# B&R Automation Studio project Agroittica (part 5)

#### Cyclic.st
```iecst
PROGRAM _CYCLIC

	//data to write
	kgb:=0;

	FOR kgb := 0 TO kgb < 30 DO
		rpt_row[kgb]:= 1;
	END_FOR;

	IF (NOT glb_data.Trigger) THEN  rpt_write_req := 0; END_IF

	IF (fucking_debug) THEN step_rpt := step_force; END_IF

	//comando reset progressivo
	IF (struct_time.day <> Saved_day (*Day_test<> Saved_day*)) THEN
		Counter_Reset := 1;
	END_IF;

	CASE step_rpt OF (* Stato di idle *)
		WAIT:
			TP_01.IN := 0;
			IF (glb_data.Trigger AND (NOT rpt_write_req))THEN

				xxx 				:= 0;
				step_rpt 			:= CHECK_FILES_NAME;
				rpt_write_req 		:= 1;				// Resetto la richiesta di scrittura del report
				glb_data.Trigger 	:= 0;			// Machine Cycle done Trigger reset;

				TP_01.IN := 1;

			END_IF
		ERROR:

			IF (glb_data.Trigger AND (NOT rpt_write_req))THEN

				xxx 				:= 0;
				step_rpt 			:= CHECK_FILES_NAME;
				rpt_write_req 		:= 1;				// Resetto la richiesta di scrittura del report
				glb_data.Trigger 	:= 0;			// Machine Cycle done Trigger reset;

			END_IF

		CHECK_FILES_NAME:	// GUARDO SE IL FILE CREATO E' LO STESSO DEL MASTER

			step_rpt := CREATE_FILE_NAME;

		CREATE_FILE_NAME: 	// CREO IL NOME DEI FILE

			memset (ADR(FileCreate_01),         0, SIZEOF(FileCreate_01)	);
			memset (ADR(FileWrite_01),          0, SIZEOF(FileWrite_01) 	);
			memset (ADR(FileClose_01),          0, SIZEOF(FileClose_01) 	);
			memset (ADR(FileCreate_03),         0, SIZEOF(FileCreate_03)    );
			memset (ADR(FileOpen_03),           0, SIZEOF(FileOpen_03)      );
			memset (ADR(FileWrite_03),          0, SIZEOF(FileWrite_03)     );
			memset (ADR(FileClose_03),          0, SIZEOF(FileClose_03)		);
			memset (ADR(string_rpt),			0, SIZEOF(string_rpt)		);
			memset (ADR(nome_file_doc),			0, SIZEOF(nome_file_doc)	);
			memset (ADR(nome_file_csv),			0, SIZEOF(nome_file_csv)	);
			memset (ADR(support_str),			0, SIZEOF(support_str)		);
			offset 		:= 0;

			(* Trasferisco nella struttura support_str l'orario attuale *)
			DT_TO_DTStructure(glb_time, ADR(struct_time));

			(* Genero il nome del file con la data odierna formato YYYY-MM-DD *)

			// inserimento anno nel nome del file
			memset (ADR(support_str), 0, SIZEOF(support_str));
			itoa(struct_time.year, ADR(support_str));
			strcpy(ADR(nome_file_doc), ADR(support_str));
			strcat(ADR(nome_file_doc), ADR(space));

			// inserimento mese nel nome del file
			memset (ADR(support_str), 0, SIZEOF(support_str));
			itoa(struct_time.month, ADR(support_str));
			IF (strlen(ADR(support_str)) = 1) THEN strcat(ADR(nome_file_doc), ADR("0")); END_IF;
			strcat(ADR(nome_file_doc), ADR(support_str));
			strcat(ADR(nome_file_doc), ADR(space));

			// inserimento giorno nel nome del file
			memset (ADR(support_str), 0, SIZEOF(support_str));
			itoa(struct_time.day, ADR(support_str));
			(*itoa(Day_test, ADR(support_str));*)
			IF (strlen(ADR(support_str)) = 1) THEN strcat(ADR(nome_file_doc), ADR("0")); END_IF;
			strcat(ADR(nome_file_doc), ADR(support_str));
			strcat(ADR(nome_file_doc), ADR(space));

			//Reset del numero progressivo quando cambia giorno
			IF Counter_Reset THEN
				Counter := 0;
				Counter_Reset := 0;
			END_IF;

			//inserimento del numero progressivo alla fine del nome del file csv
			memset (ADR(support_str), 0, SIZEOF(support_str));
			itoa(Counter, ADR(support_str));
			IF (strlen(ADR(support_str)) = 1) THEN strcat(ADR(nome_file_doc), ADR("0")); END_IF;
			strcat(ADR(nome_file_doc), ADR(support_str));

			strcpy(ADR(nome_file_csv), ADR(nome_file_doc));
			strcat(ADR(nome_file_csv), ADR(estensione));				// creo il file YYYY-MM-DD.csv

			step_rpt := CREATE_CSV_FILE;

		CREATE_CSV_FILE: // CREO IL FILE .CSV

			FileCreate_03.enable  := 1;
			FileCreate_03.pDevice := ADR(DATA);
			FileCreate_03.pFile   := ADR(nome_file_csv);

			FileCreate_03;

			IF (FileCreate_03.status = 0) THEN

				offset 					:= 0;
				step_rpt   				:= OPEN_CSV_FILE;
				FileCreate_03.enable 	:= 0;
				RowCounterFile			:= 0;

			ELSIF (FileCreate_03.status = 20705) THEN (* file già esistente *)
				step_rpt 				:= OPEN_CSV_FILE;
				FileCreate_03.enable 	:= 0;
			END_IF

		OPEN_CSV_FILE: // APRO IL FILE CSV

			FileOpen_03.enable    := 1;
			FileOpen_03.pDevice   := ADR(DATA);
			FileOpen_03.pFile     := ADR(nome_file_csv);
			FileOpen_03.mode      := FILE_RW;

			FileOpen_03;

			IF (FileOpen_03.status = 0) THEN

				step_rpt := CREATE_HEADER_CSV_FILE;

				memset (ADR(string_rpt), 	0, SIZEOF(string_rpt)	);
				memset (ADR(support_str),   0, SIZEOF(support_str)  );

				ident_csv			:= FileOpen_03.ident;
				FileOpen_03.enable 	:= 0;
				filelen := FileOpen_03.filelen;

			ELSIF (FileOpen_03.status <> 65535) THEN

				step_rpt	 		:= ERROR;
				numero_errore   	:= FileIoGetSysError();
				FileOpen_03.enable 	:= 0;
			END_IF

			// salvo il giorno in una variabile ritentiva
			Saved_day := struct_time.day;
			//Saved_day := Day_test;

			//Gestione numero progressivo, ogni 400000 elementi il progressivo avanza
			IF (filelen >= 400000) THEN
				New_CSV := 1;
			ELSE
				New_CSV := 0;
			END_IF;

			IF (New_CSV AND (NOT New_CSV_cmd)) THEN
				Counter 	:= Counter +1;
				New_CSV_cmd := 1;
			ELSIF ((NOT New_CSV) AND New_CSV_cmd) THEN
				New_CSV_cmd := 0;
			END_IF;

		CREATE_HEADER_CSV_FILE:

			// Il file è vuoto
			IF (filelen < 101) THEN //lunghezza della intestazione

				memset (ADR(string_rpt), 0, SIZEOF(string_rpt));
				// HEADER CDV FILE -------------------------------------------------------------------
				// Salvo l'intestazione di 120 caratteri

				//	sep:=;
				//	Report
				//	Dati misurazione particolari
				//	Mould Code := jhgfdsasdfghj;
				//
				//	Timestamp;Recipe Name;QRCode;Dato 1;Dato 2;Dato 3;Dato 4;Dato 5;Dato 6;Dato 7;Dato 8;Code;Material type;Material Color;Mould Code;Density;Volume;Peso;Temperature;Peso inserto;\n
				//  Timestamp;Recipe Name;QRCode;Dato 1;Dato 2;Dato 3;Dato 4;Dato 5;Dato 6;Dato 7;Dato 8;Code;Material type;Material Color;Mould Code;Density;Volume;Peso;Temperature;Peso inserto;\n
				//  012345678901234567890123456789012345678901234567890123456789012345678901234567890123456789012345678901234567890123456789
				//	0_________1_________2_________3_________4_________5_________6_________7_________8_________9_________10________11________

				strcpy(ADR(string_rpt), ADR('sep:=;$r$nReport$r$nDati misurazione particolari$r$n$r$n'));
				strcat(ADR(string_rpt), ADR('$r$n'));
				strcat(ADR(string_rpt), ADR('TIMESTAMP;BILANCIA;SENSORE PISTOLA;PISTONE SOLLEVAMENTO SU;PISTONE SOLLEVAMENTO GIU;PISTOLA 1;PISTOLA 2;'));
				strcat(ADR(string_rpt), ADR('$r$n'));
				// END HEADER ------------------------------------------------------------------------

				// TIMESTAMP
				memset (ADR(support_str), 0, SIZEOF(support_str));
				ascDT(glb_data.time_stamp[xxx],ADR(support_str),SIZEOF(support_str));
				IF (strlen(ADR(support_str)) = 1) THEN strcat(ADR(string_rpt), ADR('0')); END_IF
				strcat(ADR(string_rpt), ADR(support_str));
				strcat(ADR(string_rpt), ADR(';'));

				// BILANCIA
				memset (ADR(support_str), 0, SIZEOF(support_str));
				strcat(ADR(string_rpt), ADR(glb_data.bilancia[xxx]));
				strcat(ADR(string_rpt), ADR(';'));

				// SENSORE PISTOLA
				memset (ADR(support_str), 0, SIZEOF(support_str));
				itoa(glb_data.sensore_pistola[xxx], ADR(support_str));
				strcat(ADR(string_rpt), ADR(support_str));
				strcat(ADR(string_rpt), ADR(';'));

				// PISTONE SOLLEVAMENTO SU
				memset (ADR(support_str), 0, SIZEOF(support_str));
				itoa(glb_data.pistone_soll_su[xxx], ADR(support_str));
				strcat(ADR(string_rpt), ADR(support_str));
				strcat(ADR(string_rpt), ADR(';'));

				// PISTONE SOLLEVAMENTO GIU
				memset (ADR(support_str), 0, SIZEOF(support_str));
				itoa(glb_data.pistone_soll_giu[xxx], ADR(support_str));
				strcat(ADR(string_rpt), ADR(support_str));
				strcat(ADR(string_rpt), ADR(';'));

				// PISTOLA 1
				memset (ADR(support_str), 0, SIZEOF(support_str));
				itoa(glb_data.pistone_pistola_1[xxx], ADR(support_str));
				strcat(ADR(string_rpt), ADR(support_str));
				strcat(ADR(string_rpt), ADR(';'));

				// PISTOLA 2
				memset (ADR(support_str), 0, SIZEOF(support_str));
				itoa(glb_data.pistone_pistola_2[xxx], ADR(support_str));
				strcat(ADR(string_rpt), ADR(support_str));
				strcat(ADR(string_rpt), ADR(';'));

				strcat(ADR(string_rpt), ADR('$r$n'));

				filelen := 0;
				str_lenght := strlen(ADR(string_rpt)); (* restituisce la lunghezza della stringa senza terminatore nullo *)

				(* Preparo la struttura per la funzione di scrittura *)
				FileWrite_03.enable   := 1;
				FileWrite_03.ident    := ident_csv;
				FileWrite_03.offset   := filelen;
				FileWrite_03.pSrc     := ADR(string_rpt);
				FileWrite_03.len      := str_lenght;
				offset                := SIZEOF(USINT) * 240;

				RowCounterFile		  := 2; //2 ROWS * 110 BYTES
				filelen := filelen + str_lenght;

				step_rpt := WRITE_CSV_FILE;

			ELSIF (filelen > 102) THEN // Il file è già stato scritto

				memset (ADR(string_rpt), 0, SIZEOF(string_rpt));

				// TIMESTAMP
				memset (ADR(support_str), 0, SIZEOF(support_str));
				ascDT(glb_data.time_stamp[xxx],ADR(support_str),SIZEOF(support_str));
				IF (strlen(ADR(support_str)) = 1) THEN strcat(ADR(string_rpt), ADR('0')); END_IF
				strcat(ADR(string_rpt), ADR(support_str));
				strcat(ADR(string_rpt), ADR(';'));

				// BILANCIA
				memset (ADR(support_str), 0, SIZEOF(support_str));
				strcat(ADR(string_rpt), ADR(glb_data.bilancia[xxx]));
				strcat(ADR(string_rpt), ADR(';'));

				// SENSORE PISTOLA
				memset (ADR(support_str), 0, SIZEOF(support_str));
				itoa(glb_data.sensore_pistola[xxx], ADR(support_str));
				strcat(ADR(string_rpt), ADR(support_str));
				strcat(ADR(string_rpt), ADR(';'));

				// PISTONE SOLLEVAMENTO SU 1
				memset (ADR(support_str), 0, SIZEOF(support_str));
				itoa(glb_data.pistone_soll_su[xxx], ADR(support_str));
				strcat(ADR(string_rpt), ADR(support_str));
				strcat(ADR(string_rpt), ADR(';'));

				// PISTONE SOLLEVAMENTO GIU 1
				memset (ADR(support_str), 0, SIZEOF(support_str));
				itoa(glb_data.pistone_soll_giu[xxx], ADR(support_str));
				strcat(ADR(string_rpt), ADR(support_str));
				strcat(ADR(string_rpt), ADR(';'));

				// PISTOLA 1
				memset (ADR(support_str), 0, SIZEOF(support_str));
				itoa(glb_data.pistone_pistola_1[xxx], ADR(support_str));
				strcat(ADR(string_rpt), ADR(support_str));
				strcat(ADR(string_rpt), ADR(';'));

				// PISTOLA 2
				memset (ADR(support_str), 0, SIZEOF(support_str));
				itoa(glb_data.pistone_pistola_2[xxx], ADR(support_str));
				strcat(ADR(string_rpt), ADR(support_str));
				strcat(ADR(string_rpt), ADR(';'));

				strcat(ADR(string_rpt), ADR('$r$n'));

				RowCounterFile := RowCounterFile + 1;
//				filelen := RowCounterFile * 120;
//				filelen := FileOpen_03.filelen;

				str_lenght := strlen(ADR(string_rpt)); (* restituisce la lunghezza della stringa senza terminatore nullo *)

				(* Preparo la struttura per la funzione di scrittura *)
				FileWrite_03.enable   := 1;
				FileWrite_03.ident    := ident_csv;
				FileWrite_03.offset   := filelen;
				FileWrite_03.pSrc     := ADR(string_rpt);
				FileWrite_03.len      := str_lenght;
				offset                := offset + (SIZEOF(USINT) * 120);

				filelen := filelen + str_lenght;

				step_rpt := WRITE_CSV_FILE;

			ELSE  // Chiamato dal controllo densità con numero di ciclo a 0

				step_rpt := CLOSE_CSV_FILE;
			END_IF

		WRITE_CSV_FILE:

			FileWrite_03;

			IF (FileWrite_03.status = 0) THEN
				glb_data.Report_recorded 		:= 1;
				step_rpt 						:= CLOSE_CSV_FILE;
				FileWrite_03.enable 		  	:= 0;

				IF (xxx < 199) THEN
					xxx := xxx + 1;
					step_rpt 			:= CREATE_HEADER_CSV_FILE;

					//					glb_data.Trigger := 0;
				END_IF

			ELSIF (FileWrite_03.status <> 65535) THEN

				step_rpt	 		:= CLOSE_CSV_FILE;
				numero_errore   	:= FileIoGetSysError();
				FileWrite_03.enable := 0;
			END_IF

		CLOSE_CSV_FILE:

			FileClose_03.enable := 1;
			FileClose_03.ident  := ident_csv;
			FileClose_03;

			IF (FileClose_03.status = 0) THEN

//				step_rpt 				:= WAIT;
				FileClose_03.enable := 0;

			ELSIF (FileClose_03.status = 20721) THEN
				step_rpt 				:= WAIT;
				FileClose_03.enable := 0;

//				glb_data.Trigger := 1;

//				IF (xxx < 199) THEN
//					xxx := xxx + 1;
//					step_rpt 			:= OPEN_CSV_FILE;
//
////					glb_data.Trigger := 0;
//				END_IF

			ELSIF (FileClose_03.status <> 65535 AND FileClose_03.status <> 65534) THEN

				step_rpt	 		:= ERROR;

				numero_errore   	:= FileIoGetSysError();
				FileClose_03.enable := 0;
			END_IF

	END_CASE;

	(*********************************************** CREATE DIR WHERE SAVE THE CAVITIES INFO LINKE TO THE RECIPES **************************************************)

	IF ((DirCreate_05.status = 0) OR (DirCreate_05.status = 20725)) THEN	    (* IF status ok (0) OR dir already exists (20725)		 	*)
		DirCreate_05.enable 	:= 0;
	END_IF

	TP_01;

END_PROGRAM
```

#### Init.st
```iecst
PROGRAM _INIT
	(*/* Pulisco la memoria */*)

	memset (ADR(DirCreate_03),			 0, SIZEOF(DirCreate_03)   	 );
	memset (ADR(DirCreate_05),			 0, SIZEOF(DirCreate_05)   	 );
	memset (ADR(FileCreate_01),          0, SIZEOF(FileCreate_01)  	 );
	memset (ADR(FileCreate_03),          0, SIZEOF(FileCreate_03)  	 );
	memset (ADR(FileOpen_03),            0, SIZEOF(FileOpen_03)    	 );
	memset (ADR(FileWrite_01),           0, SIZEOF(FileWrite_01)   	 );
	memset (ADR(FileWrite_03),           0, SIZEOF(FileWrite_03)   	 );
	memset (ADR(FileClose_01),           0, SIZEOF(FileClose_01)	 );
	memset (ADR(FileClose_03),           0, SIZEOF(FileClose_03)	 );
	memset (ADR(string_rpt),			 0, SIZEOF(string_rpt)	 	 );
	memset (ADR(support_str),			 0, SIZEOF(support_str)  	 );

	step_rpt 			 := WAIT;
	RowCounterFile		 := 0;

	DirCreate_03.enable  := 1;
	DirCreate_03.pDevice := ADR(CF);
	DirCreate_03.pName   := ADR(DATA);

	DirCreate_03;

	IF ((DirCreate_03.status = 0) OR  (DirCreate_03.status = 20725)) THEN	    (*/* IF status ok (0) OR dir already exists (20725)			*/*)

		//DirCreate_03.status := 0;												(*/* set status ok											*/*)
	END_IF

	DirCreate_05.enable  := 1;
	DirCreate_05.pDevice := ADR(CF);
	DirCreate_05.pName   := ADR(CFG);

	DirCreate_05;

	IF ((DirCreate_05.status = 0) OR  (DirCreate_05.status = 20725)) THEN	    (*/* IF status ok (0) OR dir already exists (20725)	 		*/*)

		//DirCreate_05.status := 0;												(*/* set status ok											*/*)
	END_IF

END_PROGRAM
```

### Program Logical/main/Time

#### Variables.var
```iecst
VAR
	DTGetTime_0 : DTGetTime := (0);
	TON_FASToff : TON_10ms := (0);
END_VAR
```

#### Cyclic.ld
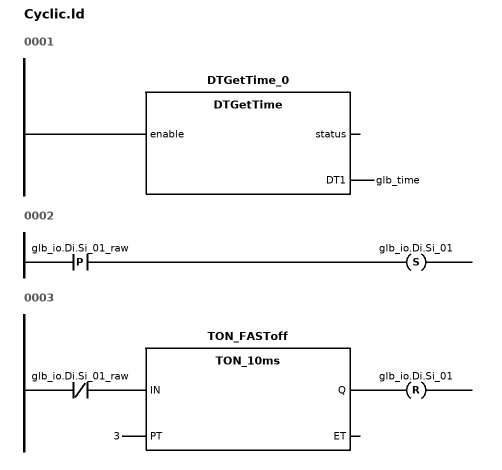
Ladder, written as Structured Text:
```iecst
PROGRAM _CYCLIC
VAR
    _e1 : R_TRIG;
END_VAR
(* Network 1 *)
DTGetTime_0(enable := TRUE);
glb_time := DTGetTime_0.DT1;

(* Network 2 *)
_e1(CLK := glb_io.Di.Si_01_raw);
IF _e1.Q THEN glb_io.Di.Si_01 := TRUE; END_IF;

(* Network 3 *)
TON_FASToff(IN := NOT glb_io.Di.Si_01_raw, PT := 3);
IF TON_FASToff.Q THEN glb_io.Di.Si_01 := FALSE; END_IF;
END_PROGRAM
```

### Program Logical/MpPkg/Recipe (IEC)

#### Variables.var
```iecst
VAR
	MpRecipeUI_0 : MpRecipeUI;
	MpRecipeRegPar_0 : MpRecipeRegPar;
	MpRecipeXml_0 : MpRecipeXml;
	UIConnect : MpRecipeUIConnectType;
	UISetup : MpRecipeUISetupType;
END_VAR
```

#### Cyclic.ld
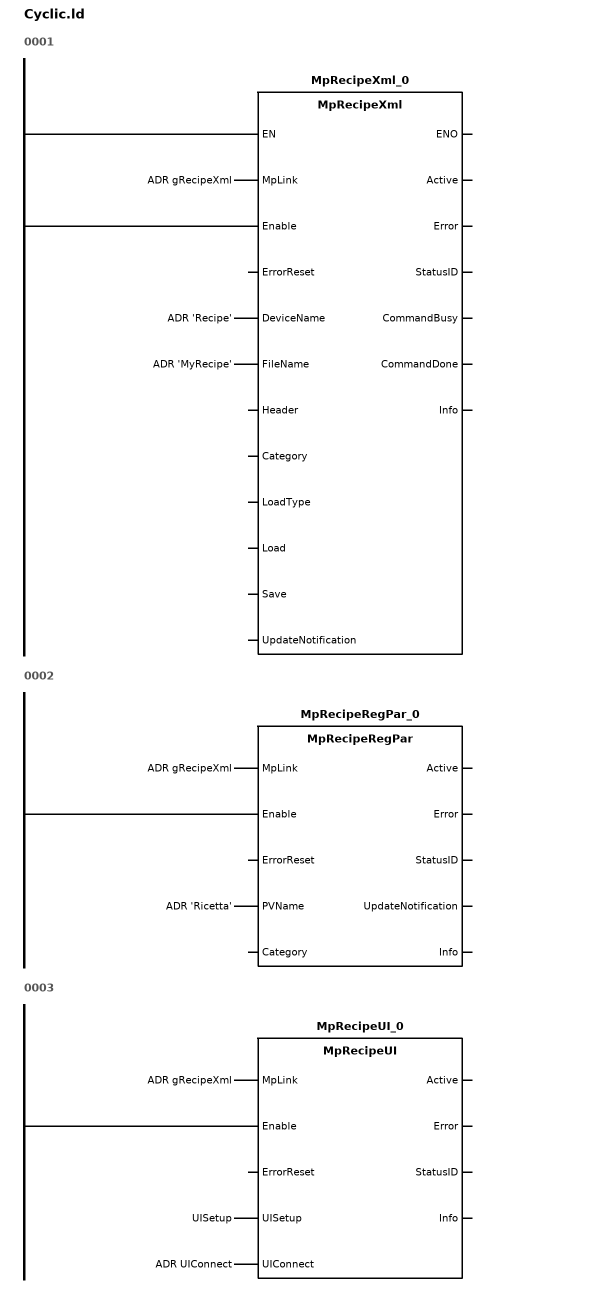
Ladder, written as Structured Text:
```iecst
PROGRAM _CYCLIC
(* Network 1 *)
MpRecipeXml_0(MpLink := ADR(gRecipeXml), Enable := TRUE, DeviceName := ADR('Recipe'), FileName := ADR('MyRecipe'));

(* Network 2 *)
MpRecipeRegPar_0(MpLink := ADR(gRecipeXml), Enable := TRUE, PVName := ADR('Ricetta'));

(* Network 3 *)
MpRecipeUI_0(MpLink := ADR(gRecipeXml), Enable := TRUE, UISetup := UISetup, UIConnect := ADR(UIConnect));
END_PROGRAM
```

### Program Logical/MpPkg/Alarm_0 (IEC)

#### Variables.var
```iecst
VAR
	avvio : BOOL;
	UserAlarm : BOOL;
	AckUserStatus : BOOL;
	AlarmXResetStatus : DINT;
	AlarmXAckStatus : DINT;
	MpAlarmXCore_0 : MpAlarmXCore;
	MpAlarmXHistory_0 : MpAlarmXHistory;
	MpAlarmXListUI_0 : MpAlarmXListUI;
	MpAlarmXListUIConnect : MpAlarmXListUIConnectType;
	AlarmXSetStatus : UDINT;
	MpAlarmXHistoryUI_0 : MpAlarmXHistoryUI;
	MpAlarmXHistoryUIConnect : MpAlarmXHistoryUIConnectType;
	XCoreEn : BOOL;
END_VAR
```

#### Cyclic.ld
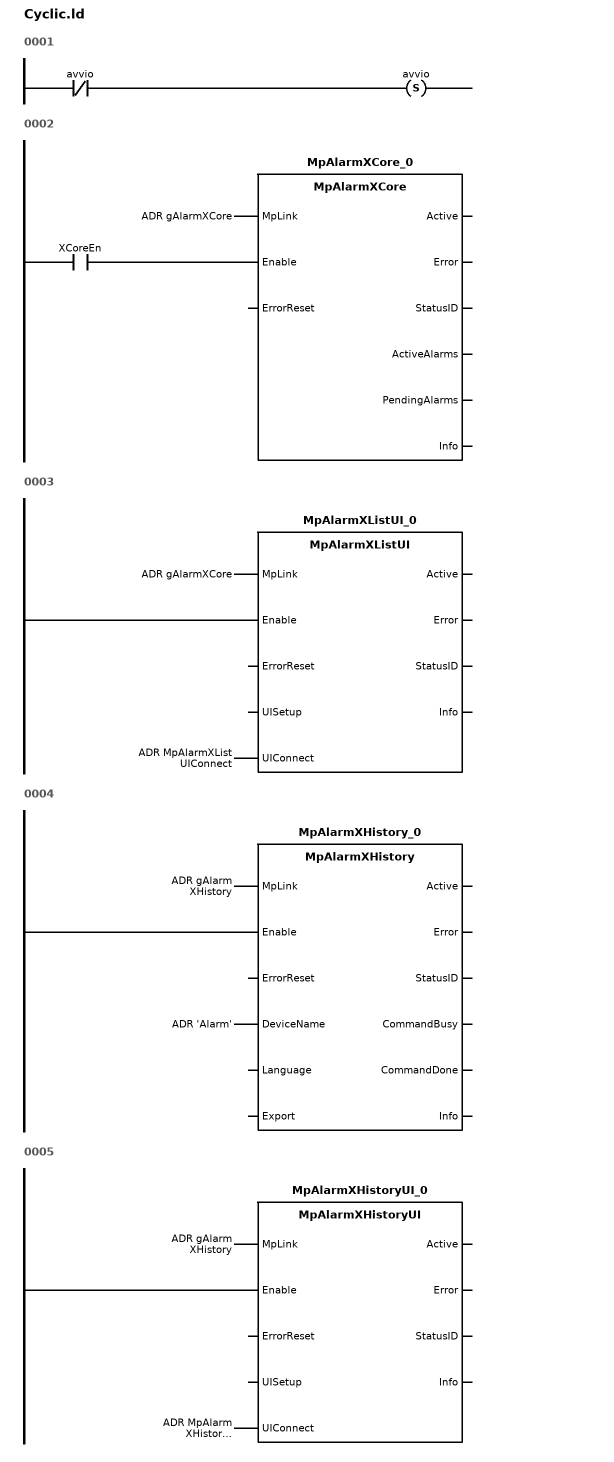
Ladder, written as Structured Text:
```iecst
PROGRAM _CYCLIC
(* Network 1 *)
IF NOT avvio THEN avvio := TRUE; END_IF;

(* Network 2 *)
MpAlarmXCore_0(MpLink := ADR(gAlarmXCore), Enable := XCoreEn);

(* Network 3 *)
MpAlarmXListUI_0(MpLink := ADR(gAlarmXCore), Enable := TRUE, UIConnect := ADR(MpAlarmXListUIConnect));

(* Network 4 *)
MpAlarmXHistory_0(MpLink := ADR(gAlarmXHistory), Enable := TRUE, DeviceName := ADR('Alarm'));

(* Network 5 *)
MpAlarmXHistoryUI_0(MpLink := ADR(gAlarmXHistory), Enable := TRUE, UIConnect := ADR(MpAlarmXHistoryUIConnect));
END_PROGRAM
```

#### Exit.ld
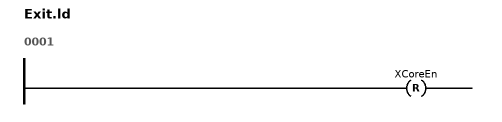
Ladder, written as Structured Text:
```iecst
PROGRAM _EXIT
(* Network 1 *)
XCoreEn := FALSE;
END_PROGRAM
```

#### Init.ld
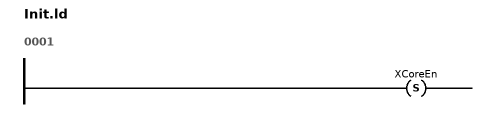
Ladder, written as Structured Text:
```iecst
PROGRAM _INIT
(* Network 1 *)
XCoreEn := TRUE;
END_PROGRAM
```

### Program Logical/MpPkg/Login

#### Variables.var
```iecst
VAR
	MpUserLoginUI_0 : MpUserLoginUI := (0);
	MpUserLogin_0 : MpUserLogin := (0);
END_VAR
```

#### Cyclic.ld
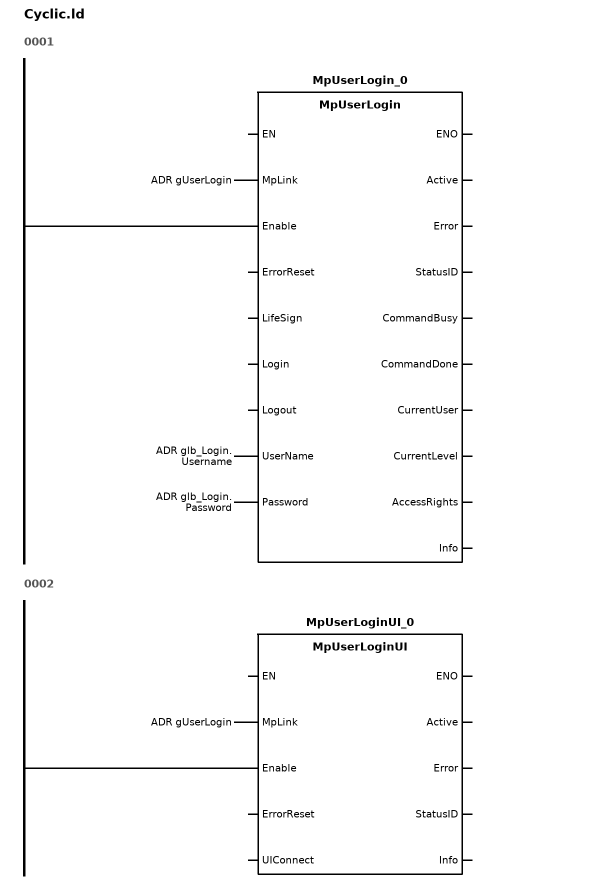
Ladder, written as Structured Text:
```iecst
PROGRAM _CYCLIC
(* Network 1 *)
MpUserLogin_0(MpLink := ADR(gUserLogin), Enable := TRUE, UserName := ADR(glb_Login.Username), Password := ADR(glb_Login.Password));

(* Network 2 *)
MpUserLoginUI_0(MpLink := ADR(gUserLogin), Enable := TRUE);
END_PROGRAM
```

### Program Logical/Allarmi/Allarm

#### Cyclic.st
```iecst
PROGRAM _CYCLIC
	(* Insert code here *)

	CASE Allarm_0.St_allarm OF

		0: //START
			IF ( Status = AUTO OR Status = MANUAL) THEN
				Allarm_0.St_allarm := 10;
			END_IF;

		10: //IDLE
			IF (glb_err.Drive1) THEN
				Allarm_0.St_allarm := 30100; //allarme M1
			END_IF;

			IF (glb_err.Drive2) THEN
				Allarm_0.St_allarm := 30200; // allarme M2
			END_IF;

			IF (glb_err.PLC) THEN
				Allarm_0.St_allarm := 30300; // allarme Fungo
			END_IF;

			IF (glb_err.Air) THEN
				Allarm_0.St_allarm := 30400; // allarme aria
			END_IF;

			IF (glb_err.Fish) THEN
				Allarm_0.St_allarm := 30500; // allarme pesce
			END_IF;

		30100: //allarme M1

			(*Status := ERR;*)
			glb_err.pending_alarms := glb_err.pending_alarms + 1;

			IF (Allarm_0.Ack) THEN
				Allarm_0.St_allarm := 40000;
			END_IF;

		30200: // allarme M2

			(*Status := ERR;*)
			glb_err.pending_alarms := glb_err.pending_alarms + 1;

			IF (Allarm_0.Ack) THEN
				Allarm_0.St_allarm := 40000;
			END_IF;

		30300: // allarme Fungo

			(*Status := ERR;*)
			glb_err.pending_alarms := glb_err.pending_alarms + 1;

			IF (Allarm_0.Ack) THEN
				Allarm_0.St_allarm := 40000;
			END_IF;

		30400: // allarme aria

			(*Status := ERR;*)
			glb_err.pending_alarms := glb_err.pending_alarms + 1;

			IF (Allarm_0.Ack) THEN
				Allarm_0.St_allarm := 40000;
			END_IF;

		30500: // allarme pesce

			(*Status := ERR;*)
			glb_err.pending_alarms := glb_err.pending_alarms + 1;
			glb_io.Do.MainAllarm := 1;

			IF (Allarm_0.Ack) THEN
				Allarm_0.St_allarm := 40000;
			END_IF;

		40000:
			glb_err.pending_alarms := 0;
			glb_io.Do.MainAllarm := 0;
			Allarm_0.St_allarm := 0;

	END_CASE;

END_PROGRAM
```

### Program Logical/Encoder (IEC)

#### Cyclic.st - Cyclic code
```iecst
PROGRAM _CYCLIC
	(* Insert code here *)

	glb_enc_sta.b_enable     := 1;

	glb_enc_sta.words        := REAL_TO_DINT( pow(2, glb_enc_sta.bit_res));
	glb_enc_sta.enc_range    := (glb_enc_sta.pinion_diam * 3.14 * glb_enc_sta.enc_rev); (*/* 7 is the motor reduction */*)
	glb_enc_sta.res          := glb_enc_sta.enc_range / glb_enc_sta.words;    (*/* Resol. in [U] is worked out  */*)

	IF (glb_enc_sta.b_enable = 1) THEN

		(*/* Reads the data from the GRAY ABSOLUTE ENCODER */*)
		glb_enc_sta.gry[0]  := glb_io.Di.enc_sta_bit_00;
		glb_enc_sta.gry[1]  := glb_io.Di.enc_sta_bit_01;
		glb_enc_sta.gry[2]  := glb_io.Di.enc_sta_bit_02;
		glb_enc_sta.gry[3]  := glb_io.Di.enc_sta_bit_03;
		glb_enc_sta.gry[4]  := glb_io.Di.enc_sta_bit_04;
		glb_enc_sta.gry[5]  := glb_io.Di.enc_sta_bit_05;
		glb_enc_sta.gry[6]  := glb_io.Di.enc_sta_bit_06;
		glb_enc_sta.gry[7]  := glb_io.Di.enc_sta_bit_07;
		glb_enc_sta.gry[8]  := glb_io.Di.enc_sta_bit_08;
		glb_enc_sta.gry[9]  := glb_io.Di.enc_sta_bit_09;
		glb_enc_sta.gry[10] := glb_io.Di.enc_sta_bit_10;
		glb_enc_sta.gry[11] := glb_io.Di.enc_sta_bit_11;

		//		Sta_Gry_To_Int(&glb_enc_sta.x, glb_enc_sta.gry);

		gray_to_int_0.gry := glb_enc_sta.gry;
		glb_enc_sta.x := gray_to_int_0.x;
		gray_to_int_0;

		Int_to_vel_0;

		IF ((glb_enc_sta.x < 0) OR (glb_enc_sta.x >= glb_enc_sta.words)) THEN
			glb_enc_sta.error := 1;
		ELSE
			glb_enc_sta.error := 0;
		END_IF
	END_IF

END_PROGRAM
```

#### Variables.var - Local variables
```iecst
VAR
	gray_to_int_0 : gray_to_int := (0);
	Int_to_vel_0 : Int_to_vel := (0);
END_VAR
```

#### LocalFunctions.fun
```iecst
FUNCTION_BLOCK Int_to_vel
	VAR_INPUT
		Pos : DINT;
	END_VAR
	VAR_OUTPUT
		Vel : REAL;
	END_VAR
	VAR_INPUT
		Maxim : DINT;
	END_VAR
	VAR
		Ton_0 : TON;
		pos_b : DINT;
		pos_a : DINT;
	END_VAR
END_FUNCTION_BLOCK

{REDUND_ERROR} FUNCTION_BLOCK gray_to_int (*TODO: Add your comment here*) (*$GROUP=User,$CAT=User,$GROUPICON=User.png,$CATICON=User.png*)
	VAR_INPUT
		gry : {REDUND_UNREPLICABLE} ARRAY[0..11] OF BOOL;
	END_VAR
	VAR_OUTPUT
		x : {REDUND_UNREPLICABLE} DINT;
	END_VAR
	VAR
		i : SINT;
		bin : ARRAY[0..11] OF BOOL;
		New_Member : USINT;
	END_VAR
END_FUNCTION_BLOCK
```

#### gray_to_int.st
```iecst
(* TODO: Add your comment here *)
FUNCTION_BLOCK gray_to_int

	bin[11] := gry[11];
	i := 0;
	x := 0;

	FOR i := 10 TO 0 BY -1 DO

		bin[i] := ((bin[i+1]) XOR (gry[i]));

	END_FOR;

	FOR i := 11 TO 0 BY -1 DO

		x := x + (bin[i] * REAL_TO_DINT( pow(2, i)));

	END_FOR;

END_FUNCTION_BLOCK

FUNCTION_BLOCK Int_to_vel

	pos_b := Pos;
	Ton_0.IN := 1;

	IF (Ton_0.Q) THEN
		Ton_0.IN := 0;
		IF (pos_b >= pos_a) THEN
			Vel := (pos_b - pos_a)/0.12;
		ELSIF (pos_a > pos_b) THEN
			Vel := (pos_b + (Maxim - pos_a))/0.12;
		END_IF
		pos_a := pos_b;

	END_IF

	Ton_0;
	Ton_0.PT := T#100ms;

END_FUNCTION_BLOCK
```

### Program Logical/FIFO/FIFO (IEC)

#### Cyclic.st - Cyclic code
```iecst
PROGRAM _CYCLIC

//	FIFO_0.INOutStatus := 1;
//	FIFO_0.DataIn := Result_String_Real;
//
//	IF (Del_Var_Sens) OR (Del_Var_Shoot) THEN
//		FIFO_0.INOutStatus := 2;
//		OutData := FIFO_0.DataOut;
//	END_IF;

//	IF Status = AUTO THEN
//		TON_clear.IN := 1;
//	END_IF;

//	IF (Status <> AUTO) THEN
//		glb_data.received_data := 0;
//		FIFO_0.clear_data := 1;
//	ELSE
//		FIFO_0.clear_data := 0;
//	END_IF

	IF (glb_io.Di.Si_01) THEN glb_pesce_passato 		:= 1; END_IF;

	IF (glb_data.WeightCmdCounter) THEN TON_clear.IN 	:= 0; END_IF;

	IF (TON_clear.Q) THEN FIFO_0.clear_data 			:= 1; END_IF

	IF Status = STOP THEN FIFO_0.clear_data 			:= 1; END_IF;

	IF Status <> STOP THEN FIFO_0.clear_data 			:= 0; END_IF;

	//Contatore messaggi -1 ricevuti dalla pesa Marel

	IF glb_data.WeightCmdCounter AND Eth_connect.Marel_Weight = '$$-1$$' THEN
		Neg_Cmd := 1;
	ELSE
		Neg_Cmd := 0;
	END_IF;

	R_TRIG_06 (CLK:=Neg_Cmd);

	IF R_TRIG_06.Q THEN
		glb_data.Neg_Weight_Counter 	:= glb_data.Neg_Weight_Counter + 1;
	END_IF;

	IF glb_data.Neg_Weight_Counter = 1000000000 THEN
		glb_data.Neg_Weight_Counter := 0;
	END_IF;

	CASE in OF
		0:
			IF (glb_data.received_data) THEN
				in 							:= 10;
				glb_data.received_data 		:= 0;

				glb_String.Raw_Length 		:= LEN(Eth_connect.Marel_Weight);
				glb_String.Length 			:= glb_String.Raw_Length - 2;
				glb_String.Result 			:= MID(Eth_connect.Marel_Weight, glb_String.Length, 2);
				glb_String.Result_Real 		:= (STRING_TO_REAL(glb_String.Result));
				glb_String.Result_Real 		:= (glb_String.Result_Real * INT_TO_REAL(1000));

				FIFO_0.INWrite 				:= 1;
				FIFO_0.DataIn 				:= glb_String.Result_Real;

			END_IF
		10:
			FIFO_0.INWrite := 0;
			in := 0;

	END_CASE

	CASE out OF
		0:
			Pesi_0.Controlled_Weight := FIFO_0.DataOut;
			OutData := FIFO_0.DataOut;
			IF (glb_st_gun_wait OR glb_cmd.Clear_weight) THEN
				out 					:= 10;
				glb_st_gun_wait 		:= 0;
				glb_cmd.Clear_weight 	:= 0;
				FIFO_0.INRead 			:= 1;
			END_IF;
		10:
			FIFO_0.INRead 	:= 0;
			out 			:= 0;

	END_CASE

//	CASE glb_FIFO.FIFO_Status OF
//
//		0:	//START
//			IF (Status = AUTO AND glb_err.pending_alarms = 0) THEN
//				glb_FIFO.FIFO_Status := 10;
//			END_IF;
//
//		10:	//AUTO IDLE
//			FIFO_0.INWrite := 0;
//
//
//			IF (glb_data.received_data) THEN
//				glb_FIFO.FIFO_Status := 20;
//				glb_data.received_data := 0;
//			END_IF;
//
//			IF ((Status <> AUTO) OR (glb_err.pending_alarms <> 0)) THEN glb_FIFO.FIFO_Status := 40; END_IF;
//
//		20:	//INSERT DATA INTO BUFFER & STRING SEPARATION
//
//			//string separation
//			glb_String.Raw_Length := LEN(Eth_connect.Marel_Weight);
//
//			glb_String.Length := glb_String.Raw_Length - 2;
//
//			glb_String.Result := MID(Eth_connect.Marel_Weight, glb_String.Length, 2);
//
//			glb_String.Result_Real := (STRING_TO_REAL(glb_String.Result));
//			glb_String.Result_Real := (glb_String.Result_Real * INT_TO_REAL(1000));
//
//			IF (Ricette.use_weight AND (glb_String.Result_Real = -1000)) THEN
//				FIFO_0.INWrite := 0;
//			ELSIF (Ricette.use_weight AND ((glb_String.Result_Real <= Pesi_0.Max_Weight_A AND glb_String.Result_Real >= Pesi_0.Min_Weight_A) OR (glb_String.Result_Real <= Pesi_0.Max_Weight_B AND glb_String.Result_Real >= Pesi_0.Min_Weight_B)))THEN
//				FIFO_0.INWrite := 1;
//				glb_registered := 1;
//			ELSE
//				FIFO_0.INWrite := 1;
//			END_IF
//
//			// Insert data into buffer
////			FIFO_0.INWrite := 1;
//			FIFO_0.DataIn := glb_String.Result_Real;
//			glb_FIFO.FIFO_Status := 40;
//
//		30:	//DELETE DATA FROM BUFFER
//			FIFO_0.INRead := 1;
//			glb_FIFO.FIFO_Status := 40;
//
//		40:	//RESET & BACK TO START
//
//			glb_FIFO.FIFO_Status := 0;
//			FIFO_0.INWrite := 0;
//
//	END_CASE;

//	CASE glb_FIFO.FIFO_Status_read OF
//
//		0: glb_FIFO.FIFO_Status_read := 10;
//
//		10:	//AUTO IDLE
//			OutData := FIFO_0.DataOut;
//			FIFO_0.INRead := 0;
//			TON_sens_in.IN := 0;
//
////			IF glb_io.Di.Si_01 AND (NOT Ricette.use_weight) THEN
//			glb_FIFO.FIFO_Status_read := 30;
//
////			END_IF;
//
//		30:	//DELETE DATA FROM BUFFER
//
//			FIFO_0.INRead := 1;
//			TON_sens_in.IN := 1;
//			glb_FIFO.FIFO_Status_read := 40;
//
//		40:	//RESET & BACK TO START
//			FIFO_0.INRead := 0;
//			//			IF ((NOT glb_io.Di.Si_01) AND TON_sens_in.Q) THEN
//			IF (glb_st_gun_wait) AND (NOT Ricette.use_weight) THEN
//				glb_FIFO.FIFO_Status_read := 0;
//				glb_st_gun_wait := 0;
//				TON_sens_in.IN := 0;
//			END_IF
//
//
//	END_CASE

	FIFO_0;

	TON_sens_in;
	TON_sens_in.PT := tempo_scans;

	TON_clear;
	TON_clear.PT := T#500ms;

	R_TRIG_06;
	R_TRIG_07;

//	Pesi_0.Controlled_Weight := FIFO_0.DataOut;

	IF test_buff THEN
		glb_FIFO.FIFO_Status := 20;
		glb_FIFO.FIFO_Status_read := 30;
		test_buff := 0;
	END_IF

END_PROGRAM
```

#### Variables.var - Local variables
```iecst
VAR
	DebugString01 : STRING[80] := '';
	Repeat_cmd : BOOL := FALSE;
END_VAR
VAR RETAIN
	Prev_value : STRING[80] := '';
END_VAR
VAR
	Count_St : USINT := 0;
	Count_Cmd : BOOL := FALSE;
	Neg_Cmd : BOOL := FALSE;
	Test : BOOL := FALSE;
	out : USINT := 0;
	in : USINT := 0;
	TON_clear : TON := (0);
	test_buff : BOOL := FALSE;
END_VAR
VAR RETAIN
	tempo_scans : TIME := T#200ms; (*200*)
END_VAR
VAR
	TON_sens_in : TON := (0);
	Del_Var_Sens_Out : BOOL := FALSE;
	Del_Var_Sens : BOOL := FALSE;
	Del_Var_Shoot_Out : BOOL := FALSE;
	Del_Var_Shoot : BOOL := FALSE;
	IN_Var_Out : BOOL := FALSE;
	IN_Var : BOOL := FALSE;
	Control_Var : {REDUND_UNREPLICABLE} BOOL := FALSE;
	OutData : REAL := 0.0;
	FIFO_0 : FIFO;
END_VAR
```

#### LocalFunctions.fun
```iecst
{REDUND_ERROR} FUNCTION_BLOCK FIFO (*TODO: Add your comment here*) (*$GROUP=User,$CAT=User,$GROUPICON=User.png,$CATICON=User.png*)
	VAR_INPUT
		DataIn : {REDUND_UNREPLICABLE} REAL;
		INOutStatus : {REDUND_UNREPLICABLE} INT;
		INWrite : BOOL;
		INRead : BOOL;
		clear_data : BOOL;
	END_VAR
	VAR_OUTPUT
		DataOut : {REDUND_UNREPLICABLE} REAL;
	END_VAR
	VAR CONSTANT
		BufferMax : INT := 5;
		BufferMin : INT := 1;
	END_VAR
	VAR
		NoOfDataPoints : {REDUND_UNREPLICABLE} INT;
		Buffer : {REDUND_UNREPLICABLE} ARRAY[BufferMin..6] OF REAL;
		pIn : {REDUND_UNREPLICABLE} INT;
		pOut : {REDUND_UNREPLICABLE} INT;
		p : INT;
	END_VAR
END_FUNCTION_BLOCK
```

#### FIFO.st
```iecst
(* TODO: Add your comment here *)
FUNCTION_BLOCK FIFO

	IF (pIn = 0) 	THEN pIn	:= BufferMin; END_IF
	IF (pOut = 0) 	THEN pOut	:= BufferMin; END_IF

//	//insert data into buffer
//	IF INOutStatus = 1 THEN
//		IF pIn <= BufferMax THEN
//			Buffer[pIn] := DataIn; //insert
//			IF NoOfDataPoints < BufferMax THEN
//				NoOfDataPoints := NoOfDataPoints +1;
//			END_IF;
//			pIn := pIn +1; //set to next element
//		ELSE //buffer full, insert into first element
//			pIn := BufferMin;
//			Buffer[pIn] := DataIn;
//			IF NoOfDataPoints < BufferMax THEN
//				NoOfDataPoints := NoOfDataPoints +1;
//			END_IF;
//			//move pointer to next element
//			pIn := pIn + 1;
//		END_IF;
	//	END_IF;

	// input
	IF (INWrite) THEN
		Buffer[4] := DataIn; //insert

		IF (Buffer[BufferMax] <> 0) THEN
			Buffer[BufferMin] := 0;
			FOR pIn:=BufferMin TO BufferMax DO
				IF (Buffer[pIn] = 0) THEN
					Buffer[pIn] := Buffer[pIn+1];
					Buffer[pIn+1] := 0;
				END_IF
			END_FOR;
		END_IF

		FOR pIn:=BufferMax TO BufferMin BY -1 DO
			IF (Buffer[pIn] = 0) THEN
				Buffer[pIn] := Buffer[pIn+1];
				Buffer[pIn+1] := 0;
			END_IF
		END_FOR;
	END_IF

	// output

	IF (INRead) THEN
		Buffer[BufferMin] := 0;
		FOR pOut:=BufferMin TO BufferMax DO
			IF (Buffer[pOut] = 0) THEN
				Buffer[pOut] := Buffer[pOut+1];
				Buffer[pOut+1] := 0;
			END_IF
		END_FOR;
	END_IF

	DataOut := Buffer[BufferMin]; // out

	IF (clear_data) THEN
		FOR p:=BufferMin TO BufferMax DO
			Buffer[p] := 0;
		END_FOR;
	END_IF

//	//take out data from buffer
//	IF INOutStatus = 2 THEN
//		IF NoOfDataPoints > 0 THEN //there must be data in buffer
//			DataOut := Buffer[pOut];
//			Buffer[pOut] := 0; //set to 0 to show that the value is removed
//			NoOfDataPoints := NoOfDataPoints -1;
//			IF pOut < BufferMax THEN
//				pOut := pOut +1;
//			ELSE
//				pOut := BufferMin;
//			END_IF;
//		END_IF;
//	END_IF;

	//buffer full. last value overwritten, move pIn pointer
//	IF NoOfDataPoints >= BufferMax THEN
////		pIn := pOut;
//		pIn := 6;
//	END_IF;

END_FUNCTION_BLOCK
```

### Library Logical/FIFO/Program

#### LocalFunctions.fun
```iecst
{REDUND_ERROR} {REDUND_UNREPLICABLE} FUNCTION_BLOCK FIFO (*TODO: Add your comment here*) (*$GROUP=User,$CAT=User,$GROUPICON=User.png,$CATICON=User.png*)
	VAR_INPUT
		DataIn : {REDUND_UNREPLICABLE} REAL;
		INOutStatus : {REDUND_UNREPLICABLE} INT;
	END_VAR
	VAR_OUTPUT
		DataOut : {REDUND_UNREPLICABLE} REAL;
	END_VAR
	VAR CONSTANT
		BufferMax : INT := 5;
		BufferMin : INT := 1;
	END_VAR
	VAR
		NoOfDataPoints : {REDUND_UNREPLICABLE} INT;
		Buffer : {REDUND_UNREPLICABLE} ARRAY[BufferMin..BufferMax] OF REAL;
		pIn : {REDUND_UNREPLICABLE} INT;
		pOut : {REDUND_UNREPLICABLE} INT;
	END_VAR
END_FUNCTION_BLOCK
```

#### Cyclic.st
```iecst
PROGRAM _CYCLIC

END_PROGRAM
```

#### FIFO.st
```iecst
(* TODO: Add your comment here *)
FUNCTION_BLOCK FIFO
	//insert data into buffer
	IF INOutStatus = 1 THEN
		IF pIn <= BufferMax THEN
			Buffer[pIn] := DataIn; //insert
			IF NoOfDataPoints < BufferMax THEN
				NoOfDataPoints := NoOfDataPoints +1;
			END_IF;
			pIn := pIn +1; //set to next element
		ELSE //buffer full, insert into first element
			pIn := BufferMin;
			Buffer[pIn] := DataIn;
			//move pointer to next element
			pIn := pIn + 1;
		END_IF;
	END_IF;

	//take out data from buffer
	IF INOutStatus = 2 THEN
		IF NoOfDataPoints > 0 THEN //there must be data in buffer
			DataOut := Buffer[pOut];
			Buffer[pOut] := 0; //set to 0 to show that the value is removed
			NoOfDataPoints := NoOfDataPoints -1;
			IF pOut < BufferMax THEN
				pOut := pOut +1;
			ELSE
				pOut := BufferMin;
			END_IF;
		END_IF;
	END_IF;

	//buffer full. last value overwritten, move pIn pointer
	IF NoOfDataPoints >= BufferMax THEN
		pIn := pOut;
	END_IF;

END_FUNCTION_BLOCK
```

### Program Logical/Keys_Lights_combos/Keys_Lights (IEC)

#### Variables.var
```iecst
VAR
	TON_03_Ctrl : BOOL := FALSE;
	ERROr : BOOL := FALSE;
	Value : USINT := 0;
	TON_01 : TON := (0);
	TON_02 : TON := (0);
	TON_03 : TON := (0);
	TON_04 : TON := (0);
	TON_05 : TON := (0);
	TON_06 : TON := (0);
	TON_03_Pulse : BOOL := FALSE;
	ALLARMi : BOOL := FALSE;
	Blink_Cmd : BOOL := FALSE;
	Blink_Counter : USINT := 0;
	RESET : BOOL := FALSE;
	Homing_Control : BOOL := FALSE;
	Homing_Control_2 : BOOL := FALSE;
	Manual_Homing_Control : BOOL := FALSE;
	Manual_Homing_Control_2 : BOOL := FALSE;
	Cartridge_Unloaded_control_2 : BOOL := FALSE;
	Cartridge_Unloaded_control : BOOL := FALSE;
	Cartridge_loaded_control : BOOL := FALSE;
	Cartridge_loaded_control_2 : BOOL := FALSE;
END_VAR
```

#### Cyclic.st
```iecst
PROGRAM _CYCLIC

	//------------------------------MOVEMENT KEYs PAIRING-------------------------------

	//PAIRING OF HMI MOVEMENT VARIABLE WITH BUTTON MOVEMENT VARIABLE
	IF (NOT glb_io.Di.Start) AND (NOT glb_io.Di.Reset) AND (NOT glb_io.Di.Backward_Mag_1) AND (NOT glb_cmd.Movement_Lock) AND (NOT glb_cmd.Movement_Lock_Homing) THEN
		MM_0.MM_Avanti := glb_io.Di.Forward_Mag_1;
	END_IF;

	//PAIRING OF HMI MOVEMENT VARIABLE WITH BUTTON MOVEMENT VARIABLE
	IF (NOT glb_io.Di.Start) AND (NOT glb_io.Di.Reset) AND (NOT glb_io.Di.Forward_Mag_1) AND (NOT glb_cmd.Movement_Lock) AND (NOT glb_cmd.Movement_Lock_Homing) THEN
		MM_0.MM_Indietro := glb_io.Di.Backward_Mag_1;
	END_IF;

	//PAIRING OF HMI MOVEMENT VARIABLE WITH BUTTON MOVEMENT VARIABLE
	IF (NOT glb_io.Di.Start) AND (NOT glb_io.Di.Reset) AND (NOT glb_io.Di.Backward_Mag_2) AND (NOT glb_cmd_2.Movement_Lock) AND (NOT glb_cmd_2.Movement_Lock_Homing) THEN
		MM_2.MM_Avanti := glb_io.Di.Forward_Mag_2;
	END_IF;

	//PAIRING OF HMI MOVEMENT VARIABLE WITH BUTTON MOVEMENT VARIABLE
	IF (NOT glb_io.Di.Start) AND (NOT glb_io.Di.Reset) AND (NOT glb_io.Di.Forward_Mag_2) AND (NOT glb_cmd_2.Movement_Lock) AND (NOT glb_cmd_2.Movement_Lock_Homing) THEN
		MM_2.MM_Indietro := glb_io.Di.Backward_Mag_2;
	END_IF;

	//PAIRING OF HMI VARIABLE WITH BEACON ALARM VARIABLE
	glb_hmi.Inp.Beacon_Alarm_Lock_1 := glb_cmd.Beeper_Lock;

	glb_hmi.Inp.Beacon_Alarm_Lock_2 := glb_cmd_2.Beeper_Lock;

	//------------------------------KEY COMBINATIONS----------------------------

	//SEQUENCE TO CONFIRM BEGINNING OF RELOADING PROCEDURE, AFTER THIS THE AXIS WILL GO BACK TO HOME POSITION FOR RELOADING, AXIS 1
	IF (Status = AUTO OR Status = MANUAL) AND glb_io.Di.Reset AND lights_status.Magazine_1 = 21 THEN
		glb_cmd.Start_Reload := 1;
	END_IF;

	//SEQUENCE TO CONFIRM BEGINNING OF RELOADING PROCEDURE, AFTER THIS THE AXIS WILL GO BACK TO HOME POSITION FOR RELOADING, AXIS 2
	IF (Status = AUTO OR Status = MANUAL) AND glb_io.Di.Reset AND lights_status.Magazine_2 = 21  THEN
		glb_cmd_2.Start_Reload := 1;
	END_IF;

	//SEQUENCE TO CONFIRM THAT THE MAGAZINE IS LOADED AND THE RELOADING PROCEDURE IS COMPLETE, THE PISTOL IS READY TO SHOOT.
	IF (Status = AUTO OR Status = MANUAL) AND glb_io.Di.Forward_Mag_1 AND glb_io.Di.Backward_Mag_1 THEN
		glb_cmd.Cartridge_loaded := 1;
	END_IF;

	//SEQUENCE TO CONFIRM THAT THE MAGAZINE IS LOADED AND THE RELOADING PROCEDURE IS COMPLETE, THE PISTOL IS READY TO SHOOT.
	IF (Status = AUTO OR Status = MANUAL) AND glb_io.Di.Forward_Mag_2 AND glb_io.Di.Backward_Mag_2 THEN
		glb_cmd_2.Cartridge_loaded := 1;
	END_IF;

	//SEQUENCE TO SET THE MAGAZINE BACK TO UNLOADED, AXIS 1
	IF (Status = AUTO OR Status = MANUAL) AND glb_io.Di.Reset AND glb_io.Di.Backward_Mag_1 AND glb_cmd.Cartridge_loaded_Gun THEN
		glb_cmd.Cartridge_loaded_Gun 	:= 0;
		Cartridge_Unloaded_control		:= 1;
	END_IF;

	//SEQUENCE TO SET THE MAGAZINE BACK TO UNLOADED, AXIS 2
	IF (Status = AUTO OR Status = MANUAL) AND glb_io.Di.Reset AND glb_io.Di.Backward_Mag_2 AND glb_cmd_2.Cartridge_loaded_Gun THEN
		glb_cmd_2.Cartridge_loaded_Gun 	:= 0;
		Cartridge_Unloaded_control_2	:= 1;
	END_IF;

	//SEQUENCE TO BEGIN THE HOMING PROCEDURE, AXIS 1
	IF (Status = AUTO OR Status = MANUAL) AND glb_io.Di.Start AND glb_io.Di.Backward_Mag_1 THEN
		glb_cmd.btn_homing := 1;
	END_IF;

	//SEQUENCE TO BEGIN THE HOMING PROCEDURE, AXIS 2
	IF (Status = AUTO OR Status = MANUAL) AND glb_io.Di.Start AND glb_io.Di.Backward_Mag_2 THEN
		glb_cmd_2.btn_homing := 1;
	END_IF;

	//
	IF glb_cmd.Cartridge_loaded THEN
		glb_cmd.Cartridge_loaded_Gun 	:= 1;
		Cartridge_loaded_control 		:= 1;
	END_IF;

	//
	IF glb_cmd_2.Cartridge_loaded THEN
		glb_cmd_2.Cartridge_loaded_Gun 	:= 1;
		Cartridge_loaded_control_2		:= 1;
	END_IF;

	//--------------------------------MOVEMENT LOCKING-------------------------------

	//LOCKING MANUAL MOVEMENT WHEN AXIS ARE HOMED, UNLOCKING WHEN THE AXIS MOVEMENT WHEN THEY ARE RELOADING

		//FIRST AXIS
		IF glb_cmd.Cartridge_loaded_Gun  THEN
			glb_cmd.Movement_Lock := 1;
		ELSE
			glb_cmd.Movement_Lock := 0;
		END_IF;

		//SECOND AXIS
		IF glb_cmd_2.Cartridge_loaded_Gun THEN
			glb_cmd_2.Movement_Lock := 1;
		ELSE
			glb_cmd_2.Movement_Lock := 0;
		END_IF;

	//LOCKING AXIS MANUAL MOVEMENTS WHILE AXIS ARE HOMING

		//FIRST AXIS
		IF glb_cmd.Homing_Lock THEN
			glb_cmd.Movement_Lock_Homing := 1;
		ELSE
			glb_cmd.Movement_Lock_Homing := 0;
		END_IF;

		//SECOND AXIS
		IF glb_cmd_2.Homing_Lock THEN
			glb_cmd_2.Movement_Lock_Homing := 1;
		ELSE
			glb_cmd_2.Movement_Lock_Homing := 0;
		END_IF;

	//----------------------------------------------------------------LIGHT COMBINATIONS----------------------------------------------------------

	//----------------------------------------------------MANAGMENT OF THE START, STOP AND RESET LEDS---------------------------------------------
	CASE lights_status.Bottom OF

		0: //START
			IF (Status = AUTO OR Status = MANUAL) THEN
				glb_io.Do.Green_Light	:= 1;
				glb_io.Do.Red_Light		:= 0;
				lights_status.Bottom 	:= 10;
			ELSIF Status = STOP THEN
				glb_io.Do.Green_Light	:= 0;
				glb_io.Do.Red_Light		:= 1;
			END_IF;

			IF Status = ERR THEN lights_status.Bottom := 100; END_IF;

		10://IDLE
			Blink_Cmd := 0;

			//MAG_1 LOADED ACKNOWLEDGE
			IF Cartridge_loaded_control THEN
				lights_status.Bottom := 20;
			END_IF;

			//MAG_2 LOADED ACKNOWLEDGE
			IF Cartridge_loaded_control_2 THEN
				lights_status.Bottom := 20;
			END_IF;

			//MAG_1 UNLOADED ACKNOWLEDGE
			IF Cartridge_Unloaded_control THEN
				lights_status.Bottom := 20;
			END_IF;

			//MAG_2 UNLOADED ACKNOWLEDGE
			IF Cartridge_Unloaded_control_2 THEN
				lights_status.Bottom := 20;
			END_IF;

			//MAG_1 HOMING ACKNOWLEDGE
			IF Homing_Control THEN
				lights_status.Bottom := 20;
			END_IF;

			//MAG_2 HOMING ACKNOWLEDGE
			IF Homing_Control_2 THEN
				lights_status.Bottom := 20;
			END_IF;

			//MAG_1 BEGIN RELOADING ACKNOWLEDGE
			IF glb_cmd.Start_Reload THEN
				lights_status.Bottom := 20;
			END_IF;

			//MAG_2 BEGIN RELOADING ACKNOWLEDGE
			IF glb_cmd_2.Start_Reload THEN
				lights_status.Bottom := 20;
			END_IF;

			IF Status = STOP THEN lights_status.Bottom := 0; END_IF;

			IF Status = ERR THEN lights_status.Bottom := 100; END_IF;

		20://BOTTOM LEDs BLINKING IN ACKNOWLEDGMENT OF SUCCESFULL INPUT
			glb_io.Do.Blue_Light 	:= TON_03_Pulse;
			glb_io.Do.Green_Light 	:= TON_03_Pulse;
			glb_io.Do.Red_Light 	:= TON_03_Pulse;

			IF (TON_03_Pulse AND (NOT Blink_Cmd)) THEN
				Blink_Counter := Blink_Counter + 1;
				Blink_Cmd := 1;
			ELSIF ((NOT TON_03_Pulse) AND Blink_Cmd) THEN
				Blink_Cmd := 0;
			END_IF

			IF Blink_Counter >= 3 THEN
				lights_status.Bottom := 21;
			END_IF;

			IF Status = ERR THEN lights_status.Bottom := 100; END_IF;

		21://RESET OF BLINKING VARIABLES AND BACK TO START
			Blink_Counter 					:= 0;
			glb_io.Do.Blue_Light 			:= 0;
			glb_io.Do.Green_Light 			:= 0;
			glb_io.Do.Red_Light 			:= 0;
			Cartridge_loaded_control 		:= 0;
			Cartridge_loaded_control_2		:= 0;
			Cartridge_Unloaded_control		:= 0;
			Cartridge_Unloaded_control_2	:= 0;
			Homing_Control					:= 0;
			Homing_Control_2				:= 0;
			glb_cmd.Cartridge_loaded		:= 0;
			glb_cmd_2.Cartridge_loaded		:= 0;
			lights_status.Bottom 			:= 0;

		100://BLUE LED BLINKING WHEN THE MACHINE IS IN EMERGENCY
			glb_io.Do.Green_Light 		:= 0;
			glb_io.Do.Red_Light  		:= 1;

			Beacon_1.White				:= 0;
			Beacon_1.Green 				:= 0;
			Beacon_1.Beeper_Alarm		:= 0;
			Beacon_2.White				:= 0;
			Beacon_2.Green 				:= 0;
			Beacon_2.Beeper_Alarm		:= 0;

			glb_io.Do.Blue_Light 		:= TON_03_Pulse;

			//WHEN YOU PRESS RESET BUTTON IT RESETS ALL ACTIVE ALARMS
			IF glb_io.Di.Reset THEN
				lights_status.Bottom 	:= 110;
			END_IF;

		110://RESET OF BLUE LED & BACK TO START

			glb_io.Do.Blue_Light 		:= 0;
			glb_io.Do.Green_Light 		:= 0;
			glb_err.pending_alarms 		:= 0;
			lights_status.Bottom		:= 0;

	END_CASE;

	//---------------------------------------------MANAGMENT OF THE BEACON LIGHTS AND BEEPER, AXIS 1----------------------------------------------
	CASE lights_status.Magazine_1 OF

		0://START
			IF (Status = AUTO OR Status = MANUAL) THEN
				lights_status.Magazine_1 	:= 10;
			END_IF;

		10://IDLE

			//Set Magazine loaded at first start up
			IF Cartridge_loaded_control THEN
				lights_status.Magazine_1 	:= 15;
			END_IF;

			//Set Magazine unloaded
			IF Cartridge_Unloaded_control THEN
				lights_status.Magazine_1 	:= 16;
			END_IF;

			//RELOAD NEEDED
			IF Empty_Mag_1_0.Empty_Mag_Sensor THEN
				lights_status.Magazine_1 	:= 20;
			END_IF;

			//AXIS NOT HOMED
			IF (NOT glb_axis_1_homed) THEN
				lights_status.Magazine_1 	:= 30;
			END_IF

			IF Status = STOP THEN lights_status.Magazine_1 := 0; END_IF;

			IF Status = ERR THEN lights_status.Magazine_1 := 0; END_IF;

		15://Set Green Beacon on, magazine loaded
			Beacon_1.Green 				:= 1;
			Beacon_1.White 				:= 0;
			Beacon_1.Beeper_Alarm 		:= 0;
			Cartridge_loaded_control 	:= 0;
			lights_status.Magazine_1 	:= 0;

		16://Set White beacon flashing, magazine unloaded
			Beacon_1.Green 				:= 0;
			Beacon_1.White 				:= TON_03_Pulse;
			Beacon_1.Beeper_Alarm 		:= 0;
			(*lights_status.Magazine_1 	:= 0;*)

			IF glb_cmd.Cartridge_loaded THEN
				lights_status.Magazine_1 := 23;
			END_IF;

		20://REOAD LIGHTS PROCEDURE, WHITE BEACON AND BLUE LED BILNKING, BUZZER BEEPS ONLY 3 TIMES
			Beacon_1.Green 			:= 0;

			Beacon_1.White 			:= TON_03_Pulse;
			(*Beacon_1.Beeper_Alarm 	:= TON_03_Pulse;*) //IT DOESN'T FUCKING BEEP
			glb_io.Do.Blue_Light 	:= TON_03_Pulse;

			IF (TON_03_Pulse AND (NOT Blink_Cmd)) THEN
				Blink_Counter := Blink_Counter + 1;
				Blink_Cmd := 1;
			ELSIF ((NOT TON_03_Pulse) AND Blink_Cmd) THEN
				Blink_Cmd := 0;
			END_IF;

			IF Blink_Counter >= 3 THEN
				lights_status.Magazine_1 := 21;
			END_IF;

			IF Status = STOP THEN Beacon_1.Beeper_Alarm := 0; lights_status.Magazine_1 := 0; END_IF;

			IF Status = ERR THEN Beacon_1.Beeper_Alarm := 0; lights_status.Magazine_1 := 0; END_IF;

		21://WHITE BEACON BLINKING AND BLUE LED BLINKING, BEACON BUZZER STOP

			Beacon_1.Beeper_Alarm 		:= 0;

			Beacon_1.White 				:= TON_03_Pulse;
			glb_io.Do.Blue_Light		:= TON_03_Pulse;

			//PRESS RESET TO SWITCH OFF BLUE BLINKING LED AND START RELOADING MOVEMENT
			IF glb_io.Di.Reset THEN
				lights_status.Magazine_1 := 22;
			END_IF;

			IF Status = STOP THEN lights_status.Magazine_1 := 0; END_IF;

			IF Status = ERR THEN lights_status.Magazine_1 := 0; END_IF;

		22://ONLY WHITE BEACON FLASHING
			glb_io.Do.Blue_Light := 0;

			Beacon_1.White := TON_03_Pulse;

			IF glb_cmd.Cartridge_loaded THEN
				lights_status.Magazine_1 := 23;
			END_IF;

		23://RESET & BACK TO START, GREEN BEACON ON
			Beacon_1.Green 				:= 1;
			Beacon_1.White 				:= 0;
			Beacon_1.Beeper_Alarm 		:= 0;
			glb_cmd.Beeper_Lock			:= 0;
			lights_status.Magazine_1	:= 0;

		30://GREEN AND WHITE BEACON BLINKING IF AXIS IS NOT HOMED
			IF (NOT glb_axis_1_homed) THEN
				Beacon_1.White 			:= TON_03_Pulse;
				Beacon_1.Green			:= TON_03_Pulse;
			END_IF

			//AXIS HOMED
			IF glb_axis_1_homed THEN
				lights_status.Magazine_1 := 31;
			END_IF;

			IF Status = STOP THEN lights_status.Magazine_1 := 0; END_IF;

			IF Status = ERR THEN lights_status.Magazine_1 := 0; END_IF;

		31://RESET AFTER AXIS HOMED
			Beacon_1.Green 				:= 0;
			Beacon_1.White 				:= 0;
			lights_status.Magazine_1 	:= 0;

	END_CASE;

	//----------------------------------------------MANAGMENT OF THE BEACON LIGHT AND BEEPER, AXIS 2------------------------------------------
	CASE lights_status.Magazine_2 OF

		0://START
			IF (Status = AUTO OR Status = MANUAL) THEN
				lights_status.Magazine_2 	:= 10;
			END_IF;

		10://IDLE

			//Set Magazine loaded at first start up
			IF Cartridge_loaded_control_2 THEN
				lights_status.Magazine_2 	:= 15;
			END_IF;

			//Set Magazine unloaded
			IF Cartridge_Unloaded_control_2 THEN
				lights_status.Magazine_2 	:= 16;
			END_IF;

			//RELOAD NEEDED
			IF Empty_Mag_22.Empty_Mag_Sensor THEN
				lights_status.Magazine_2 	:= 20;
			END_IF;

			//AXIS NOT HOMED
			IF (NOT glb_axis_2_homed)	THEN
				lights_status.Magazine_2 	:= 30;
			END_IF;

			IF Status = ERR THEN lights_status.Magazine_2 := 0; END_IF;

		15:
			Beacon_2.Green 				:= 1;
			Beacon_2.White 				:= 0;
			Beacon_2.Beeper_Alarm 		:= 0;
			lights_status.Magazine_2 	:= 0;

		16:
			Beacon_2.Green 				:= 0;
			Beacon_2.White 				:= TON_03_Pulse;
			Beacon_2.Beeper_Alarm 		:= 0;
			(*lights_status.Magazine_2 	:= 0;*)

			IF glb_cmd_2.Cartridge_loaded THEN
				lights_status.Magazine_2 := 23;
			END_IF;

		20://REOAD LIGHTS PROCEDURE, WHITE BEACON AND BLUE LED BILNKING, BEEPER BEEPS ONLY 3 TIMES
			Beacon_2.Green			:= 0;

			Beacon_2.White 			:= TON_03_Pulse;
			glb_io.Do.Blue_Light 	:= TON_03_Pulse;
			(*Beacon_2.Beeper_Alarm 	:= TON_03_Pulse;*) //IT DOESN'T FUCKING BEEP pt.2

			IF (TON_03_Pulse AND (NOT Blink_Cmd)) THEN
				Blink_Counter 	:= Blink_Counter + 1;
				Blink_Cmd 		:= 1;
			ELSIF ((NOT Beacon_2.Beeper_Alarm) AND Blink_Cmd) THEN
				Blink_Cmd 		:= 0;
			END_IF;

			IF Blink_Counter >= 3 THEN
				lights_status.Magazine_2 := 21;
			END_IF;

			IF Status = ERR THEN lights_status.Magazine_2 := 0; END_IF;

		21://WHITE BEACON BLINKING
			Beacon_2.Beeper_Alarm		:= 0;
			Beacon_1.White 				:= TON_03_Pulse;
			glb_io.Do.Blue_Light		:= TON_03_Pulse;

			//PRESS RESET TO SWITCH OFF BLUE BLINKING LED AND START RELOAD MOVEMENT
			IF glb_io.Di.Reset THEN
				lights_status.Magazine_1 := 22;
			END_IF;

			IF Status = STOP THEN lights_status.Magazine_2 := 0; END_IF;

			IF Status = ERR THEN lights_status.Magazine_2 := 0; END_IF;

		22:
			Beacon_2.White				:= TON_03_Pulse;

			IF glb_cmd_2.Cartridge_loaded THEN
				lights_status.Magazine_1 := 23;
			END_IF;

			IF Status = ERR THEN lights_status.Magazine_2 := 0; END_IF;

		23://RESET & BACK TO START, GREEN BEACON ON
			Beacon_2.Green 				:= 1;
			Beacon_2.White 				:= 0;
			Beacon_2.Beeper_Alarm 		:= 0;
			Cartridge_loaded_control_2 	:= 0;
			lights_status.Magazine_2	:= 0;

		30://GREEN AND WHITE BEACON BLINKING IF AXIS IS NOT HOMED
			IF (NOT glb_axis_2_homed) THEN
				Beacon_2.Green := TON_03_Pulse;
				Beacon_2.White := TON_03_Pulse;
			END_IF;

			//AXIS HOMED
			IF glb_axis_2_homed THEN
				lights_status.Magazine_2 := 31;
			END_IF;

			IF Status = ERR THEN lights_status.Magazine_2 := 0; END_IF;

		31://RESET AFTER AXIS HOMED
			Beacon_2.Green 				:= 0;
			Beacon_2.White 				:= 0;
			lights_status.Magazine_2 	:= 0;

	END_CASE;

	//---------------------------------TIMERS----------------------------------

	TON_03;
	TON_04;

	TON_03( IN:=NOT TON_04.Q, PT:=T#0.5s);
	TON_03_Pulse := TON_03.Q;

	TON_04( IN:=TON_03.Q, PT:= T#0.5s);

END_PROGRAM
```

### Program Logical/RT/Program (ReAction)

- Cyclic.rti - Cyclic code (not shown)

### Program Logical/Sim

#### Variables.var
```iecst
VAR
	Debugstring2 : STRING[80] := '';
	Debugstring1 : STRING[80] := '';
	Debugstring : STRING[80] := '';
	fish_cmd : USINT := 0;
	tempo_del_cazzo : USINT := 0;
	Second_Scan : USINT := 0;
	random1 : UDINT := 0;
	random : UDINT := 0;
	ton_0 : TON := (0);
	ton_1 : TON := (0);
	ton_3 : TON := (0);
	TP_01 : TP := (0);
	TON_06 : TON := (0);
	ton_2 : TON := (0);
	time_2 : TIME := T#500ms;
	time_1 : TIME := T#500ms;
	time_ms : TIME := T#0S;
	time_0 : TIME := T#0S;
	support_str : STRING[40];
	bilancia_simulata : REAL := 0.250;
	diminuisci : BOOL := FALSE;
	random_send : BOOL := FALSE;
	START_Fish : BOOL := FALSE;
	STOP_fish : BOOL := FALSE;
END_VAR
```

#### Cyclic.st
```iecst
PROGRAM _CYCLIC

	IF Simu_enable THEN

		//set variabili per simulazione
		glb_err_sim.Drive1 			:= 0;

		glb_err_sim.Drive2 			:= 0;

		glb_err_sim.pending_alarms 	:= 0;

		glb_err_sim.Air				:= 0;

		glb_err_sim.Em_Bt			:= 0;

		//simulatore nastro pesci
		CASE fish_cmd OF

			0:
				IF START_Fish AND (NOT STOP_fish) THEN
					fish_cmd := 10;
				END_IF;

			10:
				TON_06.IN := 1;

				IF TON_06.Q = 1 THEN
					fish_cmd := 20;
				END_IF;

				IF STOP_fish THEN
					fish_cmd := 30;
				END_IF;

			20:
				glb_io.Di.Si_01 := 1;
				Debugstring		:='on';
				fish_cmd		:= 30;

			30:
				glb_io.Di.Si_01 := 0;
				Debugstring1	:='off';
				TON_06.IN		:= 0;
				fish_cmd 		:= 0;

		END_CASE;

		//Timer

		TON_06;

		TON_06.PT := T#750ms;

		TP_01;

		TP_01.PT := T#1s;

		//Pairing segnali per simulazione
		glb_io.Di.Start 			:= glb_io_sim.Di.Start;

		glb_io.Di.Stop 				:= glb_io_sim.Di.Stop;

		glb_io.Di.Automatic 		:= glb_io_sim.Di.Automatic;

		glb_io.Di.Manual 			:= glb_io_sim.Di.Manual;

		glb_io.Di.Reset				:= glb_io_sim.Di.Reset;

		glb_io.Di.Forward_Mag_1		:= glb_io_sim.Di.Forward_Mag_1;

		glb_io.Di.Backward_Mag_1	:= glb_io_sim.Di.Backward_Mag_1;

		glb_io.Di.Forward_Mag_2		:= glb_io_sim.Di.Forward_Mag_2;

		glb_io.Di.Backward_Mag_2	:= glb_io_sim.Di.Backward_Mag_2;

		glb_err.Drive1 				:= glb_err_sim.Drive1;

		glb_err.Drive2 				:= glb_err_sim.Drive2;

		glb_err.pending_alarms 		:= glb_err_sim.pending_alarms;

		glb_err.Air					:= glb_err_sim.Air;

		glb_err.Em_Bt				:= glb_err_sim.Em_Bt;

	END_IF;

END_PROGRAM
```

#### Init.st
```iecst
PROGRAM _INIT
	(* Insert code here *)
	time_ms := clock_ms();
	time_0 := time_ms;
	time_1 := time_ms + T#500ms;
	time_2 := time_1;

END_PROGRAM
```

### Program Logical/XSM_Demo_vnc/xsm_demo (IEC) - A new program

#### xsm_demo.var - Local variables
```iecst
(********************************************************************
 * COPYRIGHT -- Bernecker + Rainer
 ********************************************************************
 * Program: ramp_sg4
 * File: ramp_sg4.var
 * Author: leesa
 * Created: March 27, 2009
 ********************************************************************
 * Local variables of program ramp_sg4
 ********************************************************************)
VAR
	Res_abs_pos : BOOL := FALSE;
	Auto_Homing_Ack : BOOL := FALSE;
	CMD_Reboot_pos : BOOL := FALSE;
	CMD_Reboot_pos_status : USINT := 0;
	Actual_Position_0 : UDINT := 0;
	old_pos : DINT := 0;
	Motor_state : En_status := STOP;
END_VAR
VAR RETAIN
	posizione_salvata : DINT := 0;
END_VAR
VAR
	init_motor_complete : BOOL := FALSE;
	CMD_home_status : USINT := 0;
	Homed : BOOL := FALSE;
	motor_init : BOOL := FALSE;
	Init_motor_status : USINT := 0;
	Dim_etichetta : DINT := 7;
	FW_step_status : USINT := 0;
	Homing_status : USINT := 0;
	limit_bypass : USINT := 0;
	XSM_Ctrl_0 : XSM_Ctrl := (0);
	XSM_IO_Cfg_0 : XSM_IO_Cfg := (0);
	XSM_AcyclicRead_0 : XSM_AcyclicRead := (0);
END_VAR
```

#### xsm_demo.st - Implementation code
```iecst
(********************************************************************
 * COPYRIGHT -- Bernecker + Rainer
 ********************************************************************
 * Program: xsm_demo
 * File: xsm_demo.st
 * Author: leesa
 * Created: July 24, 2009
 ********************************************************************
 * Implementation of program xsm_demo
 ********************************************************************)

PROGRAM _INIT

	IF (posizione_salvata <> 0) THEN Actual_Position_0 := posizione_salvata; END_IF;

	(* Set up XSM Control parameters. *)
	XSM_Ctrl_0.IO_Mapping.DeviceName := 'IF6.ST2';					(* Location of SM module on X20 CPU. *)
	XSM_Ctrl_0.IO_Mapping.Channel := 1;								(* Channel number, motor 1 on the module. *)

	XSM_Ctrl_0.Parameters.Units_rev := 700;							(* User scaling, units per rev. *)
	XSM_Ctrl_0.Parameters.PosSWLimit := 100000;						(* Units based on user scaling, change to suit application. *)
	XSM_Ctrl_0.Parameters.NegSWLimit := -100;						(* Units based on user scaling, change to suit application. *)
	XSM_Ctrl_0.Parameters.HomePosition := 0;						(* Units based on user scaling, change to suit application. *)
	XSM_Ctrl_0.Parameters.HomeMode := 0;							(* Required homing mode, change to suit application. *)
	XSM_Ctrl_0.Parameters.Ignore_SWLimits := FALSE;					(* On. *)
	XSM_Ctrl_0.Parameters.Ignore_HWLimits := FALSE;					(* On. *)
	XSM_Ctrl_0.Parameters.HWLimits_Active_Low := FALSE;				(* Off. *)
	XSM_Ctrl_0.Parameters.StallDetectionEnable := FALSE;			(* Off. *)
	XSM_Ctrl_0.Parameters.UnderCurrentDetectionEnable := FALSE;		(* Off. *)

	(* Set up I/O configuration - No need to defind in AS I/O Configuration for module. *)
	XSM_IO_Cfg_0.IO_Cfg.MixedDecayCfg := 15;							(* AS Default, change to suit application. *)

	XSM_IO_Cfg_0.IO_Cfg.Current.Holding := 1.5;							(* A, Change to suit motor/application. *)
	XSM_IO_Cfg_0.IO_Cfg.Current.Rated := 1.5;							(* A, Change to suit motor/application. *)
	XSM_IO_Cfg_0.IO_Cfg.Current.Maximum := 2.0; 						(* A, Change to suit motor/application. *)

	XSM_IO_Cfg_0.IO_Cfg.FullStepThreshold := 0;							(* Also sets to AS Default of 65535, change to suit application. *)

	XSM_IO_Cfg_0.IO_Cfg.StallCfg.StallDetection := 0;					(* AS Default, change to suit application. *)
	XSM_IO_Cfg_0.IO_Cfg.StallCfg.StallDetection := FALSE;				(* AS Default, change to suit application. *)

	XSM_IO_Cfg_0.IO_Cfg.RefCfg.ReferencingConfiguration := 0;			(* AS Default (Positive edge 0 ), change to suit application. *)
	XSM_IO_Cfg_0.IO_Cfg.RefCfg.StallRecongnitionDelay := 8;				(* AS Default units of 25ms, change to suit application. *)

	XSM_IO_Cfg_0.IO_Cfg.MPGen.MaxSpeed :=			1000;					(* Units/s based on user scaling, change to suit application. *)
	XSM_IO_Cfg_0.IO_Cfg.MPGen.MaxAcc :=				5000;					(* Units/s/s based on user scaling, change to suit application. *)
	XSM_IO_Cfg_0.IO_Cfg.MPGen.MaxDec :=				5000;					(* Units/s/s based on user scaling, change to suit application. *)
	XSM_IO_Cfg_0.IO_Cfg.MPGen.RevLoop := 			0;						(* Units based on user scaling, change to suit application. *)
	XSM_IO_Cfg_0.IO_Cfg.MPGen.FixedPos_a :=			0;						(* Units based on user scaling, change to suit application. *)
	XSM_IO_Cfg_0.IO_Cfg.MPGen.FixedPos_b :=			0;						(* Units based on user scaling, change to suit application. *)
	XSM_IO_Cfg_0.IO_Cfg.MPGen.RefSpeed :=			100;					(* Units/s based on user scaling, change to suit application. *)
	XSM_IO_Cfg_0.IO_Cfg.MPGen.JoltTimeLimitation:=	0;						(* AS Default, change to suit application. *)

	XSM_IO_Cfg_0.pIO_Mapping := ADR(XSM_Ctrl_0.IO_Mapping);				(* Pass IO mapping structure from XSM_Ctrl(). *)
	XSM_IO_Cfg_0.pParameters := ADR(XSM_Ctrl_0.Parameters);				(* Pass parameter structure from XSM_Ctrl(). *)

	(* Set up AcyclicRead(). *)
	XSM_AcyclicRead_0.pIO_Mapping :=	ADR(XSM_Ctrl_0.IO_Mapping);		(* Pass IO mapping structure from XSM_Ctrl(). *)

END_PROGRAM

PROGRAM _CYCLIC

	(* ONLY FOR DEMO PURPOSES WITH VCN & SG4 OR WATCH & SGC. *)
	(* You need to make required state machine and error handling for your application. *)

	//2023 - SET VARIABLES OF SECOND FUNCTION BLOCK

	Module_OK := XSM_Ctrl_0.IO_Mapping.ModuleOK;
	Module_ID := XSM_Ctrl_0.IO_Mapping.ModuleID;
	Input_Status := XSM_Ctrl_0.IO_Mapping.InputStatus;

	XSM_Ctrl_0(); (* Call function. *)
	XSM_IO_Cfg_0(); (* Call function. *)
	XSM_AcyclicRead_0(); (* Call function. *)

	XSM_Ctrl_0.Cmd.Reset := glb_hmi.Out.Reset;

	glb_err.Drive1 := XSM_Ctrl_0.Error;

	//---------------------------------KEY PAIRING---------------------------------

	//PAIRING OF AUTO HOMING ACK BUTTON

	Auto_Homing_Ack := glb_cmd.Auto_Homing_Ack;

	//PAIRING OF RESET BUTTON

	XSM_Ctrl_0.Cmd.Reset := glb_io.Di.Reset;

	//MOD FOR HOMING AND LIGHT CONTROL

	First_Homing := Homed;

	glb_axis_1_homed := Homed;

	//PAIRING FOR MOVEMENT KEY LOCKING WHILE ONGOING HOMING PROCEDURE

	glb_cmd.Homing_Lock := Homing_status <> 0;

	//-------------------------------------------------------------------------------------------------

	IF (Status <> ERR) THEN XSM_Ctrl_0.Enable := TRUE; END_IF

	CASE Init_motor_status OF

		0: IF (NOT motor_init) THEN motor_init := 1; Init_motor_status := 10; END_IF

		10:
			XSM_IO_Cfg_0.Enable := TRUE;
			IF (XSM_IO_Cfg_0.Status = 0) THEN Init_motor_status := 20; END_IF

		20:
			XSM_IO_Cfg_0.Config := TRUE;
			IF (XSM_IO_Cfg_0.Done) THEN Init_motor_status := 30; END_IF

		30:
			XSM_IO_Cfg_0.Config := FALSE;
			XSM_IO_Cfg_0.Enable := FALSE;
			init_motor_complete := TRUE;
			Init_motor_status := 0;

	END_CASE

	CASE Motor_state OF

		0: // idle stop
			IF (init_motor_complete AND Status = AUTO) THEN
				Motor_state := AUTO;
			ELSIF (init_motor_complete AND Status = MANUAL) THEN
				Motor_state := MANUAL;
			ELSIF (Status = ERR OR XSM_Ctrl_0.Error) THEN
				Motor_state := ERR;
			END_IF;

		10: // auto
			XSM_Ctrl_0.Power := TRUE;
			IF (Status = STOP) THEN
				Motor_state := STOP;
				XSM_Ctrl_0.Power := FALSE;
			ELSIF (Status = ERR OR XSM_Ctrl_0.Error) THEN
				Motor_state := ERR;
			END_IF

		20: // manual
			XSM_Ctrl_0.Power := TRUE;
			IF (Status = STOP) THEN
				Motor_state := STOP;
				XSM_Ctrl_0.Power := FALSE;
			ELSIF (Status = ERR OR XSM_Ctrl_0.Error) THEN
				Motor_state := ERR;
			END_IF

		30: // error
			XSM_Ctrl_0.Power := FALSE;
			IF (Status = STOP AND (NOT XSM_Ctrl_0.Error)) THEN
				glb_err.Drive1 	:= FALSE;
				Motor_state 	:= STOP;
			END_IF

	END_CASE;

	//---------------------------------------------------------------------MANUAL MOVEMENTS OF MAGAZINE MOTOR-----------------------------------------------------------------
//	CASE MM_0.MM_status OF
//
//		0:	//Start
//			IF ((Status = MANUAL OR Status = AUTO) AND glb_err.pending_alarms = 0 AND Homed AND (NOT glb_err.Drive1)) THEN
//				MM_0.MM_status := 1;
//			END_IF;
//			XSM_Ctrl_0.Cmd.Stop 					:= FALSE;
//			XSM_Ctrl_0.Parameters.Ignore_HWLimits 	:= 0;
//			XSM_Ctrl_0.Parameters.Ignore_SWLimits 	:= 0;
//
//		1:	//Idle
//			IF (MM_0.MM_Avanti AND (NOT MM_0.MM_Indietro)) THEN
//				MM_0.MM_status := 10;
//			END_IF;
//
//			IF (MM_0.MM_Indietro AND (NOT MM_0.MM_Avanti)) THEN
//				MM_0.MM_status := 20;
//			END_IF;
//
//		10:	//Forward
//			XSM_Ctrl_0.Cmd.Velocity 				:= 200;
//			XSM_Ctrl_0.Cmd.Move_Velocity 			:= TRUE;
//			XSM_Ctrl_0.Cmd.Stop 					:= FALSE;
//			XSM_Ctrl_0.Parameters.Ignore_HWLimits 	:= 1;
//			XSM_Ctrl_0.Parameters.Ignore_SWLimits 	:= 1;
//
//			IF (NOT MM_0.MM_Avanti) THEN
//				MM_0.MM_status := 30;
//			END_IF;
//
//			IF (Empty_Mag_1_0.Empty_Mag_Sensor) THEN
//				MM_0.MM_status := 40;
//			END_IF;
//
//		20:	//Backward
//			XSM_Ctrl_0.Cmd.Velocity 				:= -200;
//			XSM_Ctrl_0.Cmd.Move_Velocity 			:= TRUE;
//			XSM_Ctrl_0.Cmd.Stop 					:= FALSE;
//			XSM_Ctrl_0.Parameters.Ignore_HWLimits 	:= 1;
//			XSM_Ctrl_0.Parameters.Ignore_SWLimits 	:= 1;
//
//			IF (NOT MM_0.MM_Indietro) THEN
//				MM_0.MM_status := 30;
//			END_IF;
//
////			IF (XSM_Ctrl_0.Monitor.Actual_Position = XSM_Ctrl_0.Parameters.HomePosition) THEN
////				MM_0.MM_status := 31;
////			END_IF;
//
//			IF (XSM_Ctrl_0.Monitor.Input_1) THEN
//				MM_0.MM_status := 41;
//			END_IF;
//
//		30:	//Reset and back to safety, if moevemnt button is released by the operator
//			XSM_Ctrl_0.Cmd.Move_Velocity 	:= FALSE;
//			XSM_Ctrl_0.Cmd.Stop 			:= TRUE;
//			old_pos 						:= XSM_Ctrl_0.Monitor.Actual_Position;
//			MM_0.MM_status 					:= 0;
//
////		31:	//Left Stop
////			XSM_Ctrl_0.Cmd.Move_Velocity := FALSE;
////			XSM_Ctrl_0.Cmd.Stop := FALSE;
////			Status := STOP;
////			MM_0.MM_status := 0;
//
//		40:	//Set parameters for StepBack after sensor touch
//			XSM_Ctrl_0.Cmd.Move_Velocity 	:= FALSE;
//			XSM_Ctrl_0.Cmd.Velocity 		:= -1000;
//			XSM_Ctrl_0.Cmd.Stop 			:= TRUE;
//			MM_0.MM_status 					:= 50;
//
//		41:	//Set parameters for StepForward after sensor touch
//			XSM_Ctrl_0.Cmd.Move_Velocity 	:= FALSE;
//			XSM_Ctrl_0.Cmd.Velocity 		:= 1000;
//			XSM_Ctrl_0.Cmd.Stop 			:= TRUE;
//			MM_0.MM_status 					:= 51;
//
//		50:	//Stepback start move
//			XSM_Ctrl_0.Cmd.Stop 			:= FALSE;
//			XSM_Ctrl_0.Cmd.Move_Velocity 	:= TRUE;
//			MM_0.MM_status 					:= 60;
//
//		51:	//Stepforward start move
//			XSM_Ctrl_0.Cmd.Stop 			:= FALSE;
//			XSM_Ctrl_0.Cmd.Move_Velocity 	:= TRUE;
//			MM_0.MM_status 					:= 61;
//
//		60:	//Stepback reset & back to start
//			IF (NOT Empty_Mag_1_0.Empty_Mag_Sensor) THEN
//				XSM_Ctrl_0.Cmd.Stop 			:= TRUE;
//				XSM_Ctrl_0.Cmd.Move_Velocity 	:= FALSE;
//				MM_0.MM_status 					:= 0;
//			END_IF;
//
//		61:	//Stepforward reset, back to start
//			IF (NOT XSM_Ctrl_0.Monitor.Input_1) THEN
//				XSM_Ctrl_0.Cmd.Stop 			:= TRUE;
//				XSM_Ctrl_0.Cmd.Move_Velocity 	:= FALSE;
//				MM_0.MM_status 					:= 0;
//			END_IF;
//
//
//
	//	END_CASE;

	CASE limit_bypass OF
		0:
			IF glb_io.Di.Start AND glb_io.Di.Reset THEN
				XSM_Ctrl_0.Parameters.Ignore_HWLimits := 1;
				XSM_Ctrl_0.Parameters.Ignore_SWLimits := 1;
				limit_bypass := 10;
			END_IF
		10:
			IF NOT (glb_io.Di.Start AND glb_io.Di.Reset) THEN
				XSM_Ctrl_0.Parameters.Ignore_HWLimits := 0;
				XSM_Ctrl_0.Parameters.Ignore_SWLimits := 0;
				limit_bypass := 0;
			END_IF

	END_CASE;

	CASE MM_0.MM_status OF

		0:	//Start
			IF ((Status = MANUAL OR Status = AUTO) AND glb_err.pending_alarms = 0 AND Homed AND (NOT glb_err.Drive1)) THEN
				MM_0.MM_status := 1;
			END_IF;

		1:	//Idle
			IF (MM_0.MM_Avanti AND (NOT MM_0.MM_Indietro)) THEN
				MM_0.MM_status := 10;
			END_IF;

			IF (MM_0.MM_Indietro AND (NOT MM_0.MM_Avanti)) THEN
				MM_0.MM_status := 20;
			END_IF;

		10:	//Forward
			XSM_Ctrl_0.Cmd.Velocity 				:= 200;
			XSM_Ctrl_0.Cmd.Move_Velocity 			:= TRUE;
			XSM_Ctrl_0.Cmd.Stop 					:= FALSE;

			IF (NOT MM_0.MM_Avanti) THEN
				MM_0.MM_status := 30;
			END_IF;

		20:	//Backward
			XSM_Ctrl_0.Cmd.Velocity 				:= -200;
			XSM_Ctrl_0.Cmd.Move_Velocity 			:= TRUE;
			XSM_Ctrl_0.Cmd.Stop 					:= FALSE;

			IF (NOT MM_0.MM_Indietro) THEN
				MM_0.MM_status := 30;
			END_IF;

		30:	//Reset and back to safety, if moevemnt button is released by the operator
			XSM_Ctrl_0.Cmd.Move_Velocity 	:= FALSE;
			XSM_Ctrl_0.Cmd.Stop 			:= TRUE;
			old_pos 						:= XSM_Ctrl_0.Monitor.Actual_Position;
			MM_0.MM_status 					:= 40;

		40: // Reset all
			XSM_Ctrl_0.Cmd.Stop 			:= FALSE;
			XSM_Ctrl_0.Cmd.Move_Velocity 	:= FALSE;
			MM_0.MM_status 					:= 0;

	END_CASE;

	//POP UP DI AUTO HOMING
//	CASE Auto_Homing_Ctrl_0.Auto_Homing_Status OF
//
//		0:	//Start
//			IF ((NOT Homed) AND Status = AUTO) THEN
//				Auto_Homing_Ctrl_0.Auto_Homing_Status := 1;
//			END_IF;
//			Auto_Homing_Ctrl_0.Pop_Up := 1;
//			Auto_Homing_Ack := 0;
//			Auto_Homing_Ctrl_0.Auto_Homing_Ack_Pop_Up := FALSE;
//
//		1:	//Pop Up
//			Auto_Homing_Ctrl_0.Pop_Up := 0;
//			Auto_Homing_Ctrl_0.Auto_Homing_Status := 10;
//
//			IF (Status <> AUTO) THEN Auto_Homing_Ctrl_0.Auto_Homing_Status := 40; END_IF;
//
//		10:	//Ack Pop Up
//			IF (Auto_Homing_Ack) THEN
//				Auto_Homing_Ctrl_0.Pop_Up := 1;
//				Auto_Homing_Ctrl_0.Auto_Homing_Status := 20;
//			END_IF;
//
//			IF (Status <> AUTO) THEN Auto_Homing_Ctrl_0.Auto_Homing_Status := 40; END_IF;
//
//		20:	//Movement
//			Auto_Homing_Ctrl_0.Auto_Homing_Ack_Pop_Up := TRUE;
//			Auto_Homing_Ctrl_0.Auto_Homing_Status := 30;
//
//			IF (Status <> AUTO) THEN Auto_Homing_Ctrl_0.Auto_Homing_Status := 40; END_IF;
//
//		30:	//Back to start
//			IF (Homed) THEN
//				Auto_Homing_Ctrl_0.Auto_Homing_Status := 40;
//			END_IF;
//
//			IF (Status <> AUTO) THEN Auto_Homing_Ctrl_0.Auto_Homing_Status := 40; END_IF;
//
//		40:
//			Auto_Homing_Ctrl_0.Auto_Homing_Status := 0;
//
//	END_CASE;

	//------------------------------------------------------------------------RELOAD MANAGEMENT---------------------------------------------------------------
	CASE Empty_Mag_1_0.Empty_Mag_Status OF

		0:	//Start
			IF (Status = AUTO AND Homed AND XSM_Ctrl_0.PowerOn AND Empty_Mag_1_0.Empty_Mag_Sensor AND glb_err.pending_alarms = 0) THEN
				glb_cmd.Cartridge_loaded_Gun 	:= 0;
				Empty_Mag_1_0.Empty_Mag_Status 	:= 10;
			END_IF;
			Empty_Mag_1_0.Empty_Mag_Pop_Up 	:= 1;
			XSM_Ctrl_0.Cmd.Move_Absolute 	:= FALSE;

		10:	//Acknowledge movement & Start Movement
			IF (glb_cmd.Start_Reload OR Empty_Mag_1_0.Empty_Mag_Ack) THEN
				glb_cmd.Start_Reload := 0;
				glb_cmd.Torna_a_casa := 1;
			END_IF;

			IF (XSM_Ctrl_0.Monitor.Actual_Position = XSM_Ctrl_0.Parameters.HomePosition OR glb_cmd.Cartridge_loaded) THEN
				Empty_Mag_1_0.Empty_Mag_Status := 11;
			END_IF;

			IF (Status <> AUTO) THEN Empty_Mag_1_0.Empty_Mag_Status := 30; END_IF;

		11:	//Operator sets magazine to loaded status
			IF (glb_cmd.Cartridge_loaded) THEN
				Empty_Mag_1_0.Empty_Mag_Status := 20;
			END_IF;

			IF (Status <> AUTO) THEN Empty_Mag_1_0.Empty_Mag_Status := 30; END_IF;

		20:	//Back to start
			Empty_Mag_1_0.Empty_Mag_Ack 	:= FALSE;
			Empty_Mag_1_0.Empty_Mag_Status 	:= 0;

	END_CASE;

	//--------------------------------------------------------------------HOMING MANAGEMENT----------------------------------------------------------------
	CASE Homing_status OF

		0: //Start
			IF (((glb_cmd.btn_homing OR Auto_Homing_Ctrl_0.Auto_Homing_Ack_Pop_Up) AND (Status = MANUAL OR Status = AUTO)) AND XSM_Ctrl_0.PowerOn) THEN
				Homing_status 		:= 1;
				glb_cmd.btn_homing 	:= 0;
			END_IF;

		1:	//Set parameters for move
			XSM_Ctrl_0.Cmd.Velocity 				:= -200;
			XSM_Ctrl_0.Cmd.Stop 					:= FALSE;
			XSM_Ctrl_0.Parameters.Ignore_SWLimits 	:= TRUE;
			XSM_Ctrl_0.Parameters.Ignore_HWLimits 	:= TRUE;
			Homing_status 							:= 10;

			IF ( Status <> MANUAL AND Status <> AUTO) THEN Homing_status:= 50; END_IF;

		10:	//Star move
			XSM_Ctrl_0.Cmd.Move_Velocity 	:= TRUE;
			Homing_status 					:= 20;

			IF ( Status <> MANUAL AND Status <> AUTO) THEN Homing_status:= 50; END_IF;

		20:	//Stop when sensor touch
			IF ((XSM_Ctrl_0.IO_Mapping.InputStatus = 1) OR (XSM_Ctrl_0.IO_Mapping.InputStatus = 3)) THEN
				XSM_Ctrl_0.Cmd.Stop 	:= TRUE;
				XSM_Ctrl_0.Cmd.Velocity := 200;
				Homing_status 			:= 30;
			END_IF;

			IF ( Status <> MANUAL AND Status <> AUTO) THEN Homing_status:= 50; END_IF;

		30:	//Step forward after sensor touch
			XSM_Ctrl_0.Cmd.Stop 			:= FALSE;
			XSM_Ctrl_0.Cmd.Move_Velocity 	:= TRUE;
			Homing_status 					:= 40;

			IF ( Status <> MANUAL AND Status <> AUTO) THEN Homing_status:= 50; END_IF;

		40: //Stop when sensor not triggered anymore
			IF (NOT (XSM_Ctrl_0.IO_Mapping.InputStatus = 1) AND NOT (XSM_Ctrl_0.IO_Mapping.InputStatus = 3)) THEN
				XSM_Ctrl_0.Cmd.Stop 	:= TRUE;
				Homing_status 			:= 50;
			END_IF;

			IF ( Status <> MANUAL AND Status <> AUTO) THEN Homing_status:= 50; END_IF;

		50: //Reset & back to start
			XSM_Ctrl_0.Cmd.Stop := FALSE;
			XSM_Ctrl_0.Cmd.Home := TRUE;
			IF (XSM_Ctrl_0.Monitor.Home_OK AND XSM_Ctrl_0.Monitor.Actual_Position = 0) THEN
				XSM_Ctrl_0.Cmd.Home 					:= FALSE;
				XSM_Ctrl_0.Cmd.Move_Velocity 			:= FALSE;
				XSM_Ctrl_0.Parameters.Ignore_SWLimits 	:= FALSE;
				XSM_Ctrl_0.Parameters.Ignore_HWLimits 	:= FALSE;
				Homed 									:= 1;
				old_pos 								:= 0;
				Homing_status 							:= 0;
				glb_cmd.Cartridge_loaded_Gun			:= 0;
			END_IF;

	END_CASE;

	//----------------------------------------------------------------AUTOMATIC FORWARD STEP----------------------------------------------------------
	CASE FW_step_status OF

		0: // start
			IF (Status = AUTO AND (NOT Empty_Mag_1_0.Empty_Mag_Sensor)) THEN FW_step_status := 1; END_IF;

		1: // idle auto
			XSM_Ctrl_0.Cmd.Distance 	:= Dim_etichetta;
			old_pos 					:= XSM_Ctrl_0.Monitor.Actual_Position;

			IF ((glb_cmd.sparo) AND XSM_Ctrl_0.PowerOn AND Homed) THEN FW_step_status := 10; glb_cmd.sparo := 0; END_IF;

			IF (Empty_Mag_1_0.Empty_Mag_Sensor) THEN FW_step_status := 20; END_IF;

			IF (Status <> AUTO) THEN FW_step_status := 20; END_IF;

		10: //automatic forward step
			XSM_Ctrl_0.Cmd.Move_Additive := TRUE;

			IF (XSM_Ctrl_0.Monitor.Actual_Position >= (old_pos + Dim_etichetta)) THEN
				old_pos 		:= XSM_Ctrl_0.Monitor.Actual_Position;
				FW_step_status 	:= 20;
			END_IF;

			IF (Empty_Mag_1_0.Empty_Mag_Sensor) THEN FW_step_status := 20; END_IF;

			IF (Status <> AUTO) THEN FW_step_status := 20; END_IF;

		20://reset & back to start
			XSM_Ctrl_0.Cmd.Move_Additive 	:= FALSE;
			FW_step_status 					:= 0;

	END_CASE;

	//---------------------------------------------------------------AUTOMATIC RETURN TO HOME POSITION-----------------------------------------------------
	CASE CMD_home_status OF
		0: // idle
			IF (Status = AUTO OR Status = MANUAL) THEN CMD_home_status := 1; END_IF

			IF (posizione_salvata <> 0) THEN Actual_Position_0 := posizione_salvata; END_IF;

		1: // idle auto

			IF (glb_cmd.Torna_a_casa AND XSM_Ctrl_0.PowerOn AND Homed) THEN
				XSM_Ctrl_0.Cmd.Position 	:= 0;
				CMD_home_status 			:= 10;
				glb_cmd.Torna_a_casa 		:= 0;
			END_IF;

			IF (Status <> AUTO AND Status <> MANUAL) THEN CMD_home_status := 60; END_IF;

		10: //start move
			Disable_refresh_pos 					:= 1;
			XSM_Ctrl_0.Cmd.Velocity 				:= -200;
			XSM_Ctrl_0.Cmd.Move_Velocity 			:= TRUE;
			XSM_Ctrl_0.Parameters.Ignore_HWLimits 	:= TRUE;
			XSM_Ctrl_0.Parameters.Ignore_SWLimits 	:= TRUE;
//			IF (XSM_Ctrl_0.Monitor.Actual_Position = 0) THEN
//				CMD_home_status := 20;
			IF (XSM_Ctrl_0.Monitor.Input_1) THEN
				CMD_home_status := 30;
			END_IF;

			IF (Status <> AUTO AND Status <> MANUAL) THEN CMD_home_status := 60; END_IF;

//		20:
//			XSM_Ctrl_0.Cmd.Move_Absolute := FALSE;
//			(*XSM_Ctrl_0.Cmd.Stop := TRUE;*)
//			old_pos := 0;
//			CMD_home_status := 0;

		30:	//stop move
			XSM_Ctrl_0.Cmd.Move_Velocity 	:= FALSE;
			XSM_Ctrl_0.Cmd.Stop 			:= TRUE;
			XSM_Ctrl_0.Cmd.Velocity 		:= 1000;
			CMD_home_status 				:= 40;

			IF (Status <> AUTO AND Status <> MANUAL) THEN CMD_home_status := 60; END_IF;

		40: //step forward
			XSM_Ctrl_0.Cmd.Stop 			:= FALSE;
			XSM_Ctrl_0.Cmd.Move_Velocity 	:= TRUE;
			IF (NOT XSM_Ctrl_0.Monitor.Input_1) THEN
				XSM_Ctrl_0.Cmd.Stop 		:= TRUE;
				CMD_home_status 			:= 50;
			END_IF;

			IF (Status <> AUTO AND Status <> MANUAL) THEN CMD_home_status := 60; END_IF;

		50: //reset & back to start
			XSM_Ctrl_0.Cmd.Move_Velocity 	:= FALSE;
			XSM_Ctrl_0.Cmd.Stop 			:= FALSE;
			XSM_Ctrl_0.Cmd.Home 			:= TRUE;
			IF (XSM_Ctrl_0.Monitor.Home_OK AND XSM_Ctrl_0.Monitor.Actual_Position = 0) THEN
				XSM_Ctrl_0.Cmd.Home 					:= FALSE;
				XSM_Ctrl_0.Cmd.Move_Velocity 			:= FALSE;
				XSM_Ctrl_0.Parameters.Ignore_SWLimits 	:= FALSE;
				XSM_Ctrl_0.Parameters.Ignore_HWLimits 	:= FALSE;
				Homed 									:= 1;
				CMD_home_status 						:= 0;
				old_pos 								:= 0;
			END_IF;

		60:
			XSM_Ctrl_0.Cmd.Move_Velocity := FALSE;
			CMD_home_status := 0;

	END_CASE;

	//-----------------------------------------------------------------------REBOOT TO PREVIOUS POSITION------------------------------------------------------

	//2024- TEST PENDING!!!!!!
	CASE CMD_Reboot_pos_status OF
		0://start
			IF (Status = AUTO OR Status = MANUAL) AND (Homed) THEN
				CMD_Reboot_pos_status := 1;
			END_IF;

			IF (posizione_salvata <> 0) THEN Actual_Position_0 := posizione_salvata; END_IF;

		1://idle
			IF (glb_cmd.Reboot_pos) THEN
				CMD_Reboot_pos_status := 2;
			END_IF;

		2://
			XSM_Ctrl_0.Cmd.Position 	:= Actual_Position_0;
			IF (XSM_Ctrl_0.PowerOn AND Homed) THEN
				CMD_Reboot_pos_status 	:= 10;
				glb_cmd.Reboot_pos 		:= 0;
			END_IF;

			IF (Status <> AUTO AND Status <> MANUAL) THEN CMD_Reboot_pos_status := 20; END_IF;

		10:
			XSM_Ctrl_0.Cmd.Move_Absolute := TRUE;

			 IF (XSM_Ctrl_0.Monitor.Actual_Position = Actual_Position_0) THEN
				old_pos 				:= XSM_Ctrl_0.Monitor.Actual_Position;
				Disable_refresh_pos 	:= 0;
				CMD_Reboot_pos_status 	:= 20;
			END_IF;

			IF (Status <> AUTO AND Status <> MANUAL) THEN CMD_Reboot_pos_status := 20; END_IF;

		20:
			XSM_Ctrl_0.Cmd.Move_Absolute := FALSE;
			CMD_Reboot_pos_status := 0;

	END_CASE;

	//MOD FOR SIMULATOR
	IF ( glb_sim = 1) THEN
//		XSM_Ctrl_0.Monitor.Actual_Position := Stepper_1_position;
	END_IF;

	IF (XSM_Ctrl_0.Monitor.Home_OK AND (NOT Disable_refresh_pos)) THEN 	posizione_salvata := XSM_Ctrl_0.Monitor.Actual_Position; END_IF;

END_PROGRAM

PROGRAM _EXIT

(* TODO : Add your code here *)

END_PROGRAM
```

#### xsm_demo_M2.st - not listed in the package file held
```iecst
(********************************************************************
 * COPYRIGHT -- Bernecker + Rainer
 ********************************************************************
 * Program: xsm_demo
 * File: xsm_demo.st
 * Author: leesa
 * Created: July 24, 2009
 ********************************************************************
 * Implementation of program xsm_demo
 ********************************************************************)

PROGRAM _INIT

	IF (posizione_salvata_2_2 <> 0) THEN Actual_position_2 := posizione_salvata_2_2; END_IF

	(* Set up XSM Control parameters. *)
	XSM_Ctrl_2.IO_Mapping.DeviceName := 'IF6.ST2';					(* Location of SM module on X20 CPU. *)
	XSM_Ctrl_2.IO_Mapping.Channel := 1;								(* Channel number, motor 1 on the module. *)

	XSM_Ctrl_2.Parameters.Units_rev := 700;							(* User scaling, units per rev. *)
	XSM_Ctrl_2.Parameters.PosSWLimit := 19000;						(* Units based on user scaling, change to suit application. *)
	XSM_Ctrl_2.Parameters.NegSWLimit := -100;						(* Units based on user scaling, change to suit application. *)
	XSM_Ctrl_2.Parameters.HomePosition := 0;						(* Units based on user scaling, change to suit application. *)
	XSM_Ctrl_2.Parameters.HomeMode := 0;							(* Required homing mode, change to suit application. *)
	XSM_Ctrl_2.Parameters.Ignore_SWLimits := FALSE;					(* On. *)
	XSM_Ctrl_2.Parameters.Ignore_HWLimits := FALSE;					(* On. *)
	XSM_Ctrl_2.Parameters.HWLimits_Active_Low := FALSE;				(* Off. *)
	XSM_Ctrl_2.Parameters.StallDetectionEnable := FALSE;			(* Off. *)
	XSM_Ctrl_2.Parameters.UnderCurrentDetectionEnable := FALSE;		(* Off. *)

	(* Set up I/O configuration - No need to defind in AS I/O Configuration for module. *)
	XSM_IO_Cfg_2.IO_Cfg.MixedDecayCfg := 15;							(* AS Default, change to suit application. *)

	XSM_IO_Cfg_2.IO_Cfg.Current.Holding := 0.20;						(* A, Change to suit motor/application. *)
	XSM_IO_Cfg_2.IO_Cfg.Current.Rated := 1.20;							(* A, Change to suit motor/application. *)
	XSM_IO_Cfg_2.IO_Cfg.Current.Maximum := 1.50;						(* A, Change to suit motor/application. *)

	XSM_IO_Cfg_2.IO_Cfg.FullStepThreshold := 0;							(* Also sets to AS Default of 65535, change to suit application. *)

	XSM_IO_Cfg_2.IO_Cfg.StallCfg.StallDetection := 0;					(* AS Default, change to suit application. *)
	XSM_IO_Cfg_2.IO_Cfg.StallCfg.StallDetection := FALSE;				(* AS Default, change to suit application. *)

	XSM_IO_Cfg_2.IO_Cfg.RefCfg.ReferencingConfiguration := 0;			(* AS Default (Positive edge 0 ), change to suit application. *)
	XSM_IO_Cfg_2.IO_Cfg.RefCfg.StallRecongnitionDelay := 8;				(* AS Default units of 25ms, change to suit application. *)

	XSM_IO_Cfg_2.IO_Cfg.MPGen.MaxSpeed :=			1000;					(* Units/s based on user scaling, change to suit application. *)
	XSM_IO_Cfg_2.IO_Cfg.MPGen.MaxAcc :=				5000;					(* Units/s/s based on user scaling, change to suit application. *)
	XSM_IO_Cfg_2.IO_Cfg.MPGen.MaxDec :=				5000;					(* Units/s/s based on user scaling, change to suit application. *)
	XSM_IO_Cfg_2.IO_Cfg.MPGen.RevLoop := 			0;						(* Units based on user scaling, change to suit application. *)
	XSM_IO_Cfg_2.IO_Cfg.MPGen.FixedPos_a :=			0;						(* Units based on user scaling, change to suit application. *)
	XSM_IO_Cfg_2.IO_Cfg.MPGen.FixedPos_b :=			0;						(* Units based on user scaling, change to suit application. *)
	XSM_IO_Cfg_2.IO_Cfg.MPGen.RefSpeed :=			100;					(* Units/s based on user scaling, change to suit application. *)
	XSM_IO_Cfg_2.IO_Cfg.MPGen.JoltTimeLimitation:=	0;						(* AS Default, change to suit application. *)

	XSM_IO_Cfg_2.pIO_Mapping := ADR(XSM_Ctrl_2.IO_Mapping);				(* Pass IO mapping structure from XSM_Ctrl(). *)
	XSM_IO_Cfg_2.pParameters := ADR(XSM_Ctrl_2.Parameters);				(* Pass parameter structure from XSM_Ctrl(). *)

	(* Set up AcyclicRead(). *)
	XSM_AcyclicRead_2.pIO_Mapping :=	ADR(XSM_Ctrl_2.IO_Mapping);		(* Pass IO mapping structure from XSM_Ctrl(). *)

END_PROGRAM

PROGRAM _CYCLIC

	(* ONLY FOR DEMO PURPOSES WITH VCN & SG4 OR WATCH & SGC. *)
	(* You need to make required state machine and error handling for your application. *)

	XSM_Ctrl_2(); (* Call function. *)
	XSM_IO_Cfg_2(); (* Call function. *)
	XSM_AcyclicRead_2(); (* Call function. *)

	XSM_Ctrl_2.Cmd.Reset := glb_hmi.Out.Reset;

	glb_err.Drive2 := XSM_Ctrl_2.Error;

	IF (Status <> ERR) THEN XSM_Ctrl_2.Enable := TRUE; END_IF

	CASE Init_motor_status_2 OF

		0: IF (NOT motor_init_2) THEN motor_init_2 := 1; Init_motor_status_2 := 10; END_IF

		10:
			XSM_IO_Cfg_2.Enable := TRUE;
			IF (XSM_IO_Cfg_2.Status = 0) THEN Init_motor_status_2 := 20; END_IF

		20:
			XSM_IO_Cfg_2.Config := TRUE;
			IF (XSM_IO_Cfg_2.Done) THEN Init_motor_status_2 := 30; END_IF

		30:
			XSM_IO_Cfg_2.Config := FALSE;
			XSM_IO_Cfg_2.Enable := FALSE;
			init_motor_complete_2 := TRUE;
			Init_motor_status_2 := 0;

	END_CASE

	CASE Motor_state_2 OF

		0: // idle stop
			IF (init_motor_complete_2 AND Status = AUTO) THEN
				Motor_state_2 := AUTO;
			ELSIF (init_motor_complete_2 AND Status = MANUAL) THEN
				Motor_state_2 := MANUAL;
			ELSIF (Status = ERR OR XSM_Ctrl_2.Error) THEN
				Motor_state_2 := ERR;
			END_IF;

		10: // auto
			XSM_Ctrl_2.Power := TRUE;
			IF (Status = STOP) THEN
				Motor_state_2 := STOP;
				XSM_Ctrl_2.Power := FALSE;
			ELSIF (Status = ERR OR XSM_Ctrl_2.Error) THEN
				Motor_state_2 := ERR;
			END_IF

		20: // manual
			XSM_Ctrl_2.Power := TRUE;
			IF (Status = STOP) THEN
				Motor_state_2 := STOP;
				XSM_Ctrl_2.Power := FALSE;
			ELSIF (Status = ERR OR XSM_Ctrl_2.Error) THEN
				Motor_state_2 := ERR;
			END_IF

		30: // error
			XSM_Ctrl_2.Power := FALSE;
			IF (Status = STOP AND (NOT XSM_Ctrl_2.Error)) THEN
				glb_err.Drive2 := FALSE;
				Motor_state_2 := STOP;
			END_IF

	END_CASE;

	CASE MM_2.MM_status OF		//Marcia Motore in manuale

		0:					//Safety check
			IF (Status = MANUAL AND glb_err.pending_alarms = 0 AND Homed_2_2 AND (NOT glb_err.Drive2)) THEN
				MM_2.MM_status := 1;
			END_IF;
			XSM_Ctrl_2.Cmd.Stop := FALSE;

		1:					//Wait for input
			IF (MM_2.MM_Avanti AND (NOT MM_2.MM_Avanti_Vel) AND (NOT MM_2.MM_Indietro) AND ( NOT MM_2.MM_Indietro_Vel)) THEN
				MM_2.MM_status := 10;
			END_IF;

			IF (MM_2.MM_Indietro AND (NOT MM_2.MM_Avanti) AND (NOT MM_2.MM_Avanti_Vel) AND ( NOT MM_2.MM_Indietro_Vel)) THEN
				MM_2.MM_status := 20;
			END_IF;

			IF (MM_2.MM_Avanti_Vel AND (NOT MM_2.MM_Avanti) AND (NOT MM_2.MM_Indietro) AND ( NOT MM_2.MM_Indietro_Vel)) THEN
				MM_2.MM_status := 11;
			END_IF;

			IF (MM_2.MM_Indietro_Vel AND (NOT MM_2.MM_Avanti) AND (NOT MM_2.MM_Indietro) AND ( NOT MM_2.MM_Avanti_Vel)) THEN
				MM_2.MM_status := 21;
			END_IF;

		10:					//Forward
			XSM_Ctrl_2.Cmd.Velocity := 200;
			XSM_Ctrl_2.Cmd.Move_Velocity := TRUE;
			XSM_Ctrl_2.Cmd.Stop := FALSE;

			IF (NOT MM_2.MM_Avanti) THEN
				MM_2.MM_status := 30;
			END_IF;

			IF (Empty_Mag_22.Empty_Mag_Sensor) THEN
				MM_2.MM_status := 40;
			END_IF;

		11:					//Fast Forward
			XSM_Ctrl_2.Cmd.Velocity := 500;
			XSM_Ctrl_2.Cmd.Move_Velocity := TRUE;
			XSM_Ctrl_2.Cmd.Stop := FALSE;

			IF (NOT MM_2.MM_Avanti_Vel) THEN
				MM_2.MM_status := 30;
			END_IF;

			IF (Empty_Mag_22.Empty_Mag_Sensor) THEN
				MM_2.MM_status := 40;
			END_IF;

		20:					//Backward
			XSM_Ctrl_2.Cmd.Velocity := -200;
			XSM_Ctrl_2.Cmd.Move_Velocity := TRUE;
			XSM_Ctrl_2.Cmd.Stop := FALSE;

			IF (NOT MM_2.MM_Indietro) THEN
				MM_2.MM_status := 30;
			END_IF;

			IF (XSM_Ctrl_2.Monitor.Actual_Position = XSM_Ctrl_2.Parameters.HomePosition) THEN
				MM_2.MM_status := 31;
			END_IF;

			IF (XSM_Ctrl_2.Monitor.Input_1) THEN
				MM_2.MM_status := 41;
			END_IF;

		21:					//Fast Backward
			XSM_Ctrl_2.Cmd.Velocity := -500;
			XSM_Ctrl_2.Cmd.Move_Velocity := TRUE;
			XSM_Ctrl_2.Cmd.Stop := FALSE;

			IF (NOT MM_2.MM_Indietro_Vel) THEN
				MM_2.MM_status := 30;
			END_IF;

		30:					//Reset and back to safety
			XSM_Ctrl_2.Cmd.Move_Velocity := FALSE;
			XSM_Ctrl_2.Cmd.Velocity := 0;
			XSM_Ctrl_2.Cmd.Stop := TRUE;
			old_pos_2_2 := XSM_Ctrl_2.Monitor.Actual_Position;
			Status := STOP;
			MM_2.MM_status := 0;

		31:					//Left Stop
			XSM_Ctrl_2.Cmd.Move_Velocity := FALSE;
			XSM_Ctrl_2.Cmd.Stop := FALSE;
			XSM_Ctrl_2.Cmd.Velocity := 0;
			Status := STOP;
			MM_2.MM_status := 0;

		40:					//StepBack after sensor touch
			XSM_Ctrl_2.Cmd.Move_Velocity := FALSE;
			XSM_Ctrl_2.Cmd.Velocity := -1000;
			XSM_Ctrl_2.Cmd.Stop := TRUE;
			MM_2.MM_status := 50;

		41:					//StepForward after sensor touch
			XSM_Ctrl_2.Cmd.Move_Velocity := FALSE;
			XSM_Ctrl_2.Cmd.Velocity := 1000;
			XSM_Ctrl_2.Cmd.Stop := TRUE;
			MM_2.MM_status := 51;

		50:					//Stepback start move
			XSM_Ctrl_2.Cmd.Stop := FALSE;
			XSM_Ctrl_2.Cmd.Move_Velocity := TRUE;
			MM_2.MM_status := 60;

		51:					//Stepforward start move
			XSM_Ctrl_2.Cmd.Stop := FALSE;
			XSM_Ctrl_2.Cmd.Move_Velocity := TRUE;
			MM_2.MM_status := 61;

		60:					//Stepback reset back to start
			IF (NOT Empty_Mag_22.Empty_Mag_Sensor) THEN
				XSM_Ctrl_2.Cmd.Stop := TRUE;
				XSM_Ctrl_2.Cmd.Move_Velocity := FALSE;
				XSM_Ctrl_2.Cmd.Velocity := 0;
				Status := STOP;
				MM_2.MM_status := 0;
			END_IF;

		61:					//Stepforward reset back to start
			IF (NOT XSM_Ctrl_2.Monitor.Input_1) THEN
				XSM_Ctrl_2.Cmd.Stop := TRUE;
				XSM_Ctrl_2.Cmd.Move_Velocity := FALSE;
				XSM_Ctrl_2.Cmd.Velocity := 0;
				Status := STOP;
				MM_2.MM_status := 0;
			END_IF;

	END_CASE;

	CASE Auto_Homing_Ctrl_2.Auto_Homing_status_2 OF  //Pop Up di Auto Homing

		0:					//Start
			IF ((NOT Homed_2) AND Status = AUTO) THEN
				Auto_Homing_Ctrl_2.Auto_Homing_status_2 := 1;
			END_IF;
			Auto_Homing_Ctrl_2.Pop_Up := 1;
			Auto_Homing_Ack_2 := 0;
			Auto_Homing_Ctrl_2.Auto_Homing_Ack_2_Pop_Up := FALSE;

		1:					//Pop Up
			Auto_Homing_Ctrl_2.Pop_Up := 0;
			Auto_Homing_Ctrl_2.Auto_Homing_status_2 := 10;

			IF (Status <> AUTO) THEN Auto_Homing_Ctrl_2.Auto_Homing_status_2 := 40; END_IF;

		10:					//Ack Pop Up
			IF (Auto_Homing_Ack_2) THEN
				Auto_Homing_Ctrl_2.Pop_Up := 1;
				Auto_Homing_Ctrl_2.Auto_Homing_status_2 := 20;
			END_IF;

			IF (Status <> AUTO) THEN Auto_Homing_Ctrl_2.Auto_Homing_status_2 := 40; END_IF;

		20:					//Movement
			Auto_Homing_Ctrl_2.Auto_Homing_Ack_2_Pop_Up := TRUE;
			Auto_Homing_Ctrl_2.Auto_Homing_status_2 := 30;

			IF (Status <> AUTO) THEN Auto_Homing_Ctrl_2.Auto_Homing_status_2 := 40; END_IF;

		30:					//Back to start
			IF (Homed_2) THEN
				Auto_Homing_Ctrl_2.Auto_Homing_status_2 := 40;
			END_IF;

			IF (Status <> AUTO) THEN Auto_Homing_Ctrl_2.Auto_Homing_status_2 := 40; END_IF;

		40:
			//Status := STOP;
			Auto_Homing_Ctrl_2.Auto_Homing_status_2 := 0;

	END_CASE;

	CASE Empty_Mag_22.Empty_Mag_Status OF      //Ricarica

		0:							//Start
			IF (Status = AUTO AND Homed_2 AND XSM_Ctrl_2.PowerOn AND Empty_Mag_22.Empty_Mag_Sensor AND glb_err.pending_alarms = 0) THEN
				Empty_Mag_22.Empty_Mag_Status := 10;
			END_IF;
			Empty_Mag_22.Empty_Mag_Pop_Up := 1;
			XSM_Ctrl_2.Cmd.Move_Absolute := FALSE;

		10:							//Pop up
			Empty_Mag_22.Empty_Mag_Pop_Up := 0;
			Empty_Mag_22.Empty_Mag_Status := 20;

			IF (Status <> AUTO) THEN Empty_Mag_22.Empty_Mag_Status := 30; END_IF;

		20:							//Pop up Ack & Start Movement
			IF (Empty_Mag_22.Empty_Mag_Ack) THEN
				glb_cmd_2.Torna_a_casa := TRUE;
				Empty_Mag_22.Empty_Mag_Pop_Up := 1;
			END_IF;

			IF (XSM_Ctrl_2.Monitor.Actual_Position = XSM_Ctrl_2.Parameters.HomePosition) THEN
				Empty_Mag_22.Empty_Mag_Status := 30;
			END_IF;

			IF (Status <> AUTO) THEN Empty_Mag_22.Empty_Mag_Status := 30; END_IF;

		30:							//Back to start
			//Status := STOP;
			old_pos_2 := 0;
			Empty_Mag_22.Empty_Mag_Ack := FALSE;
			Empty_Mag_22.Empty_Mag_Status := 0;

	END_CASE;

	CASE Homing_status_2 OF

		0:
			IF (((glb_cmd_2.btn_homing AND Status = MANUAL) OR ((NOT Homed_2) AND Status = AUTO AND Auto_Homing_Ctrl_2.Auto_Homing_Ack_2_Pop_Up)) AND XSM_Ctrl_2.PowerOn) THEN
				Homing_status_2 := 1;
				glb_cmd_2.btn_homing := 0;
			END_IF;

		1:
			XSM_Ctrl_2.Cmd.Velocity := -200;
			Homing_status_2 := 10;
			XSM_Ctrl_2.Cmd.Stop := FALSE;
			XSM_Ctrl_2.Parameters.Ignore_SWLimits := TRUE;
			XSM_Ctrl_2.Parameters.Ignore_HWLimits := TRUE;

		10:
			XSM_Ctrl_2.Cmd.Move_Velocity := TRUE;
			Homing_status_2 := 20;
		20:
			IF (XSM_Ctrl_2.IO_Mapping.InputStatus = 1) THEN
				XSM_Ctrl_2.Cmd.Stop := TRUE;
				XSM_Ctrl_2.Cmd.Velocity := 200;
				Homing_status_2 := 30;
			END_IF;
		30:
			XSM_Ctrl_2.Cmd.Stop := FALSE;
			XSM_Ctrl_2.Cmd.Move_Velocity := TRUE;
			Homing_status_2 := 40;
		40:
			IF (NOT (XSM_Ctrl_2.IO_Mapping.InputStatus = 1)) THEN
				XSM_Ctrl_2.Cmd.Stop := TRUE;
				Homing_status_2 := 50;
			END_IF;

		50:
			XSM_Ctrl_2.Cmd.Stop := FALSE;
			XSM_Ctrl_2.Cmd.Home := TRUE;
			IF XSM_Ctrl_2.Monitor.Home_OK THEN
				XSM_Ctrl_2.Cmd.Home := FALSE;
				XSM_Ctrl_2.Cmd.Move_Velocity := FALSE;
				XSM_Ctrl_2.Parameters.Ignore_SWLimits := FALSE;
				XSM_Ctrl_2.Parameters.Ignore_HWLimits := FALSE;
				Homed_2 := 1;
				Homing_status_2 := 0;
				old_pos_2 := 0;
				Status := STOP;
			END_IF;

	END_CASE;

	CASE FW_step_status_2 OF

		0: // idle
			IF (Status = AUTO AND (NOT Empty_Mag_22.Empty_Mag_Sensor)) THEN FW_step_status_2 := 1; END_IF;

		1: // idle auto
			XSM_Ctrl_2.Cmd.Distance := Dim_etichetta;
			IF ((glb_cmd_2.sparo) AND XSM_Ctrl_2.PowerOn AND Homed_2) THEN FW_step_status_2 := 10; glb_cmd_2.sparo := 0; END_IF;

			IF (Empty_Mag_22.Empty_Mag_Sensor) THEN FW_step_status_2 := 20; END_IF;

			IF (Status <> AUTO) THEN FW_step_status_2 := 20; END_IF;

		10: //
			XSM_Ctrl_2.Cmd.Move_Additive := TRUE;
			IF (XSM_Ctrl_2.Monitor.Actual_Position = (old_pos_2 + Dim_etichetta)) THEN
				old_pos_2 := XSM_Ctrl_2.Monitor.Actual_Position;
				FW_step_status_2 := 20;
			END_IF;

			IF (Empty_Mag_22.Empty_Mag_Sensor) THEN FW_step_status_2 := 20; END_IF;

			IF (Status <> AUTO) THEN FW_step_status_2 := 20; END_IF;
		20:
			XSM_Ctrl_2.Cmd.Move_Additive := FALSE;
			FW_step_status_2 := 0;

	END_CASE;

	CASE CMD_home_status_2 OF
		0: // idle
			IF (Status = AUTO OR Status = MANUAL) THEN CMD_home_status_2 := 1; END_IF

		1: // idle auto

			IF (glb_cmd_2.Torna_a_casa AND XSM_Ctrl_2.PowerOn AND Homed_2) THEN
				XSM_Ctrl_2.Cmd.Position := 0;
				CMD_home_status_2 := 10;
				glb_cmd_2.Torna_a_casa := 0;
			END_IF;

			IF (Status <> AUTO AND Status <> MANUAL) THEN CMD_home_status_2 := 21; END_IF;

		10:
			XSM_Ctrl_2.Cmd.Move_Absolute := TRUE;
			IF (XSM_Ctrl_2.Monitor.Actual_Position = 0) THEN CMD_home_status_2 := 20; END_IF;

			IF (Status <> AUTO AND Status <> MANUAL) THEN CMD_home_status_2 := 21; END_IF;

		20:
			XSM_Ctrl_2.Cmd.Move_Absolute := FALSE;
			old_pos_2 := 0;
			//Status := STOP;
			CMD_home_status_2 := 0;

		21:
			XSM_Ctrl_2.Cmd.Move_Absolute := FALSE;
			CMD_home_status_2 := 0;

	END_CASE

	CASE CMD_Reboot_pos_status_2 OF
		0: // idle
			IF (Status = AUTO OR Status = MANUAL) THEN CMD_Reboot_pos_status_2 := 1; END_IF;

		1:
			IF (glb_cmd_2.Reboot_pos) THEN CMD_Reboot_pos_status_2 := 2; END_IF;

		2: // idle auto
			XSM_Ctrl_2.Cmd.Position := Actual_position_2;
			IF (XSM_Ctrl_2.PowerOn AND Homed_2) THEN
				CMD_Reboot_pos_status_2 := 10;
				glb_cmd_2.Reboot_pos := 0;
			END_IF;

			IF (Status <> AUTO AND Status <> MANUAL) THEN CMD_Reboot_pos_status_2 := 20; END_IF;
		10:
			XSM_Ctrl_2.Cmd.Move_Absolute := TRUE;
			IF (XSM_Ctrl_2.Monitor.Actual_Position = Actual_Position_2) THEN
				old_pos_2 := XSM_Ctrl_2.Monitor.Actual_Position;
				CMD_Reboot_pos_status_2 := 20;
			END_IF;

			IF (Status <> AUTO AND Status <> MANUAL) THEN CMD_Reboot_pos_status_2 := 20; END_IF;
		20:
			XSM_Ctrl_2.Cmd.Move_Absolute := FALSE;
			CMD_Reboot_pos_status_2 := 0;

	END_CASE

	posizione_salvata_2 := XSM_Ctrl_2.Monitor.Actual_Position;

END_PROGRAM

PROGRAM _EXIT

(* TODO : Add your code here *)

END_PROGRAM
```

### Program Logical/XSM_Demo_vnc/ip_adr (IEC) - Get ip address for VCN

#### ip_adr.var - Local variables
```iecst
(********************************************************************
 * COPYRIGHT -- Bernecker + Rainer
 ********************************************************************
 * Program: ip_adr
 * File: ip_adr.var
 * Author: leesa
 * Created: July 21, 2009
 ********************************************************************
 * Local variables of program ip_adr
 ********************************************************************)
VAR
	CfgGetIPAddr_0 : CfgGetIPAddr;
	IP_Address : STRING[20];
	GetIPAddress : BOOL;
END_VAR
```

#### ip_adr.st - Implementation code
```iecst
(********************************************************************
COPYRIGHT: July 21, 2009 Bernecker + Rainer
=====================================================================

*********************************************************************)

PROGRAM _INIT

	CfgGetIPAddr_0.pDevice:= ADR('IF2');		(* X20 CPU *)

END_PROGRAM

PROGRAM _CYCLIC

	(* Get IP Address via watch required for VNC. *)
	IF (GetIPAddress = 1) THEN
		CfgGetIPAddr_0(enable := 1, pIPAddr := ADR(IP_Address), Len := 20);
		IF (CfgGetIPAddr_0.status <> ERR_FUB_BUSY) THEN
			GetIPAddress:= 0;
		END_IF
	END_IF

END_PROGRAM

PROGRAM _EXIT

(* TODO : Add your code here *)

END_PROGRAM
```

- Visualisation Logical/XSM_Demo_vnc/VGAvnc (not shown)

### Program Logical/XSM_Demo_vnc/xsm_demo_M2 (IEC) - A new program

#### xsm_demo.var - Local variables
```iecst
(********************************************************************
 * COPYRIGHT -- Bernecker + Rainer
 ********************************************************************
 * Program: ramp_sg4
 * File: ramp_sg4.var
 * Author: leesa
 * Created: March 27, 2009
 ********************************************************************
 * Local variables of program ramp_sg4
 ********************************************************************)
VAR
	glb_Auto_homing_lock : BOOL := FALSE;
	Auto_Homing_Ack_2 : BOOL := FALSE;
	CMD_Reboot_pos_2 : BOOL := FALSE;
	CMD_Reboot_pos_status_2 : USINT := 0;
	Actual_Position_2 : UDINT := 0;
	old_pos_2 : DINT := 0;
	Motor_state_2 : En_status := STOP;
END_VAR
VAR RETAIN
	posizione_salvata_2 : DINT := 0;
END_VAR
VAR
	init_motor_complete_2 : BOOL := FALSE;
	CMD_home_status_2 : USINT := 0;
	Homed_2 : BOOL := FALSE;
	motor_init_2 : BOOL := FALSE;
	Init_motor_status_2 : USINT := 0;
	Dim_etichetta : DINT := 7;
	FW_step_status_2 : USINT := 0;
	Homing_status_2 : USINT := 0;
	XSM_Ctrl_2 : XSM_Ctrl := (0);
	XSM_IO_Cfg_2 : XSM_IO_Cfg := (0);
	XSM_AcyclicRead_2 : XSM_AcyclicRead := (0);
END_VAR
```
